METHOD PRIVATE DigitalMissingImageRejected
TEST('DigitalMissingImageRejected');
trustDigitalMissingImageRejected.cfg.restoreCommandOnRestart := TRUE;
trustDigitalMissingImageRejected.cfg.invert := TRUE;
trustDigitalMissingImageRejected.SeedSavedCommand(value := FALSE);
trustDigitalMissingImageRejected.simulatedBootDataLoaded := FALSE;
trustDigitalMissingImageRejected.simulatedOldBootData := FALSE;
trustDigitalMissingImageRejected();
AssertTrue(trustDigitalMissingImageRejected.sts.outputInhibited, 'Untrusted persistent image cannot restore output');
AssertFalse(trustDigitalMissingImageRejected.outSignal, 'Electrical output honors startup trust');
trustDigitalMissingImageRejected.simulatedBootDataLoaded := TRUE; trustDigitalMissingImageRejected.simulatedOldBootData := FALSE;
trustDigitalMissingImageRejected.SimulateStartup(); trustDigitalMissingImageRejected();
AssertTrue(trustDigitalMissingImageRejected.sts.outputInhibited, 'Later trust cannot revive previously rejected saved intent');
TEST_FINISHED();
END_METHOD

METHOD PRIVATE DigitalFreshCommandWithUntrustedImage
TEST('DigitalFreshCommandWithUntrustedImage');
trustDigitalFreshCommandWithUntrustedImage.cfg.restoreCommandOnRestart := TRUE;
trustDigitalFreshCommandWithUntrustedImage.cfg.invert := TRUE;
trustDigitalFreshCommandWithUntrustedImage.SeedSavedCommand(value := FALSE);
trustDigitalFreshCommandWithUntrustedImage.simulatedBootDataLoaded := TRUE;
trustDigitalFreshCommandWithUntrustedImage.simulatedOldBootData := TRUE;
trustDigitalFreshCommandWithUntrustedImage.SetOff();
trustDigitalFreshCommandWithUntrustedImage();
AssertFalse(trustDigitalFreshCommandWithUntrustedImage.sts.outputInhibited, 'Fresh command is independent of image trust');
AssertTrue(trustDigitalFreshCommandWithUntrustedImage.outSignal, 'Electrical output honors startup trust');
trustDigitalFreshCommandWithUntrustedImage.simulatedBootDataLoaded := TRUE; trustDigitalFreshCommandWithUntrustedImage.simulatedOldBootData := FALSE;
trustDigitalFreshCommandWithUntrustedImage.SimulateStartup(); trustDigitalFreshCommandWithUntrustedImage();
AssertFalse(trustDigitalFreshCommandWithUntrustedImage.sts.outputInhibited, 'Fresh command remains valid for later trusted restoration');
TEST_FINISHED();
END_METHOD

METHOD PRIVATE AnalogBackupImageRejected
TEST('AnalogBackupImageRejected');
trustAnalogBackupImageRejected.cfg.restoreCommandOnRestart := TRUE;
trustAnalogBackupImageRejected.cfg.useRawValue := TRUE; trustAnalogBackupImageRejected.cfg.safeRaw := 17.0;
trustAnalogBackupImageRejected.SeedSavedCommand(value := 42.0);
trustAnalogBackupImageRejected.simulatedBootDataLoaded := TRUE;
trustAnalogBackupImageRejected.simulatedOldBootData := TRUE;
trustAnalogBackupImageRejected();
AssertTrue(trustAnalogBackupImageRejected.sts.outputInhibited, 'Untrusted persistent image cannot restore output');
AssertEquals_REAL(17.0, trustAnalogBackupImageRejected.sts.rawReal, 0.001, 'Analog output honors startup trust');
trustAnalogBackupImageRejected.simulatedBootDataLoaded := TRUE; trustAnalogBackupImageRejected.simulatedOldBootData := FALSE;
trustAnalogBackupImageRejected.SimulateStartup(); trustAnalogBackupImageRejected();
AssertTrue(trustAnalogBackupImageRejected.sts.outputInhibited, 'Later trust cannot revive previously rejected saved intent');
TEST_FINISHED();
END_METHOD

METHOD PRIVATE AnalogMissingImageRejected
TEST('AnalogMissingImageRejected');
trustAnalogMissingImageRejected.cfg.restoreCommandOnRestart := TRUE;
trustAnalogMissingImageRejected.cfg.useRawValue := TRUE; trustAnalogMissingImageRejected.cfg.safeRaw := 17.0;
trustAnalogMissingImageRejected.SeedSavedCommand(value := 42.0);
trustAnalogMissingImageRejected.simulatedBootDataLoaded := FALSE;
trustAnalogMissingImageRejected.simulatedOldBootData := FALSE;
trustAnalogMissingImageRejected();
AssertTrue(trustAnalogMissingImageRejected.sts.outputInhibited, 'Untrusted persistent image cannot restore output');
AssertEquals_REAL(17.0, trustAnalogMissingImageRejected.sts.rawReal, 0.001, 'Analog output honors startup trust');
trustAnalogMissingImageRejected.simulatedBootDataLoaded := TRUE; trustAnalogMissingImageRejected.simulatedOldBootData := FALSE;
trustAnalogMissingImageRejected.SimulateStartup(); trustAnalogMissingImageRejected();
AssertTrue(trustAnalogMissingImageRejected.sts.outputInhibited, 'Later trust cannot revive previously rejected saved intent');
TEST_FINISHED();
END_METHOD

METHOD PRIVATE AnalogFreshCommandWithUntrustedImage
TEST('AnalogFreshCommandWithUntrustedImage');
trustAnalogFreshCommandWithUntrustedImage.cfg.restoreCommandOnRestart := TRUE;
trustAnalogFreshCommandWithUntrustedImage.cfg.useRawValue := TRUE; trustAnalogFreshCommandWithUntrustedImage.cfg.safeRaw := 17.0;
trustAnalogFreshCommandWithUntrustedImage.SeedSavedCommand(value := 42.0);
trustAnalogFreshCommandWithUntrustedImage.simulatedBootDataLoaded := TRUE;
trustAnalogFreshCommandWithUntrustedImage.simulatedOldBootData := TRUE;
trustAnalogFreshCommandWithUntrustedImage.SetValue(rValue := 42.0);
trustAnalogFreshCommandWithUntrustedImage();
AssertFalse(trustAnalogFreshCommandWithUntrustedImage.sts.outputInhibited, 'Fresh command is independent of image trust');
AssertEquals_REAL(42.0, trustAnalogFreshCommandWithUntrustedImage.sts.rawReal, 0.001, 'Analog output honors startup trust');
trustAnalogFreshCommandWithUntrustedImage.simulatedBootDataLoaded := TRUE; trustAnalogFreshCommandWithUntrustedImage.simulatedOldBootData := FALSE;
trustAnalogFreshCommandWithUntrustedImage.SimulateStartup(); trustAnalogFreshCommandWithUntrustedImage();
AssertFalse(trustAnalogFreshCommandWithUntrustedImage.sts.outputInhibited, 'Fresh command remains valid for later trusted restoration');
TEST_FINISHED();
END_METHOD

END_FUNCTION_BLOCK

// ---- Testing/POUs/FB_OutputRestart_Probe.TcPOU
// Injects a previously persisted value into an otherwise fresh instance.
// This tests startup policy, NOT actual TwinCAT persistent-image durability.
FUNCTION_BLOCK FB_OutputRestart_Probe EXTENDS TcForge.FB_DigitalOutput
VAR_INPUT
    simulatedBootDataLoaded : BOOL := TRUE;
    simulatedOldBootData : BOOL;
END_VAR

SUPER^();

METHOD PUBLIC SeedSavedCommand
VAR_INPUT
    value : BOOL;
END_VAR
_savedCommand := value;
_savedCommandValid := TRUE;
END_METHOD

// Policy probe: reset volatile arming only; not a runtime/persistent-image test.
METHOD PUBLIC SimulateStartup
_startup := TRUE;
_commandReceived := FALSE;
_armed := FALSE;
_forceSafe := FALSE;
_safeRequested := FALSE;
_requestSync := FALSE;
END_METHOD

METHOD PROTECTED _HasTrustedPersistentImage : BOOL
// Local probe inputs only: never mutate TwinCAT system information.
_HasTrustedPersistentImage := simulatedBootDataLoaded AND NOT simulatedOldBootData;
END_METHOD

END_FUNCTION_BLOCK

// ---- Testing/POUs/FB_AnalogOutputRestart_Probe.TcPOU
// Injects a previously persisted value into an otherwise fresh instance.
// This tests startup policy, NOT actual TwinCAT persistent-image durability.
FUNCTION_BLOCK FB_AnalogOutputRestart_Probe EXTENDS TcForge.FB_AnalogOutput
VAR_INPUT
    simulatedBootDataLoaded : BOOL := TRUE;
    simulatedOldBootData : BOOL;
END_VAR

SUPER^();

METHOD PUBLIC SeedSavedCommand
VAR_INPUT
    value : REAL;
END_VAR
_savedCommand := value;
_savedCommandValid := TRUE;
END_METHOD

// Policy probe: reset volatile arming only; not a runtime/persistent-image test.
METHOD PUBLIC SimulateStartup
_startup := TRUE;
_commandReceived := FALSE;
_armed := FALSE;
_forceSafe := FALSE;
_safeRequested := FALSE;
_requestSync := 0.0;
END_METHOD

METHOD PROTECTED _HasTrustedPersistentImage : BOOL
// Local probe inputs only: never mutate TwinCAT system information.
_HasTrustedPersistentImage := simulatedBootDataLoaded AND NOT simulatedOldBootData;
END_METHOD

END_FUNCTION_BLOCK

// ---- Testing/Tests/FB_IOQualityMonitor_Test.TcPOU
FUNCTION_BLOCK FB_IOQualityMonitor_Test EXTENDS TcUnit.FB_TestSuite
VAR
_done, _cyclicDone : BOOL;
_phase : UINT;
_stale : TcForge.FB_IOQualityMonitor;
_clock : TON;
_boundaryClock : TON;
_boundary : TcForge.FB_IOQualityMonitor;
_boundaryStarted, _boundaryDone : BOOL;
END_VAR

IF NOT _done THEN
StartupNeedsNewProducerSample();
CommunicationRecoveryNeedsNewSample();
DeviceAndInvalidSampleReject();
SequenceResetNeedsNewBaseline();
DisableRequiresReacquisition();
TimeoutConfigurationReacquires();
QualityRecoveryDoesNotRearmOutput();
EtherCATStateAndWorkingCounter();
_done := TRUE; END_IF;
CyclicFreshness();
FreshnessBoundary();

METHOD StartupNeedsNewProducerSample
VAR
fb : TcForge.FB_IOQualityMonitor;
outp : TcForge.FB_DigitalOutput;
bitIndex : INT;
mask : WORD;
END_VAR
TEST('StartupNeedsNewProducerSample');
fb(enabled := TRUE, communicationGood := TRUE, deviceGood := TRUE, sampleValid := TRUE, sampleSequence := 10);
AssertEquals_INT(Expected := 0, Actual := fb.quality, Message := 'First observed frame is only a baseline');
fb(sampleSequence := 11);
AssertEquals_INT(Expected := 2, Actual := fb.quality, Message := 'New coherent producer sample enables quality');
TEST_FINISHED();
END_METHOD

METHOD CommunicationRecoveryNeedsNewSample
VAR
fb : TcForge.FB_IOQualityMonitor;
outp : TcForge.FB_DigitalOutput;
bitIndex : INT;
mask : WORD;
END_VAR
TEST('CommunicationRecoveryNeedsNewSample');
fb(enabled := TRUE, communicationGood := TRUE, deviceGood := TRUE, sampleValid := TRUE, sampleSequence := 10); fb(sampleSequence := 11);
fb(communicationGood := FALSE);
AssertEquals_INT(Expected := 1, Actual := fb.quality, Message := 'Communication loss is immediate');
fb(communicationGood := TRUE);
AssertEquals_INT(Expected := 1, Actual := fb.quality, Message := 'Frozen sample cannot restore quality');
fb(sampleSequence := 12);
AssertEquals_INT(Expected := 2, Actual := fb.quality, Message := 'Fresh sample restores quality');
TEST_FINISHED();
END_METHOD

METHOD DeviceAndInvalidSampleReject
VAR
fb : TcForge.FB_IOQualityMonitor;
outp : TcForge.FB_DigitalOutput;
bitIndex : INT;
mask : WORD;
END_VAR
TEST('DeviceAndInvalidSampleReject');
fb(enabled := TRUE, communicationGood := TRUE, deviceGood := TRUE, sampleValid := TRUE, sampleSequence := 1); fb(sampleSequence := 2);
fb(deviceGood := FALSE);
AssertEquals_INT(Expected := 3, Actual := fb.reason, Message := 'Device fault is distinct');
fb(deviceGood := TRUE, sampleValid := FALSE, sampleSequence := 3);
AssertEquals_INT(Expected := 4, Actual := fb.reason, Message := 'Invalid frame is distinct');
fb(sampleValid := TRUE);
AssertEquals_INT(Expected := 1, Actual := fb.quality, Message := 'Previously invalid sample cannot become fresh');
fb(sampleSequence := 4);
AssertEquals_INT(Expected := 2, Actual := fb.quality, Message := 'Fresh valid update recovers');
TEST_FINISHED();
END_METHOD

METHOD SequenceResetNeedsNewBaseline
VAR
fb : TcForge.FB_IOQualityMonitor;
outp : TcForge.FB_DigitalOutput;
bitIndex : INT;
mask : WORD;
END_VAR
TEST('SequenceResetNeedsNewBaseline');
fb(enabled := TRUE, communicationGood := TRUE, deviceGood := TRUE, sampleValid := TRUE, sampleSequence := 10); fb(sampleSequence := 11);
fb(sampleSequence := 0);
AssertEquals_INT(Expected := 7, Actual := fb.reason, Message := 'Producer restart invalidates old session');
fb(); AssertEquals_INT(Expected := 1, Actual := fb.quality, Message := 'Repeated reset sequence stays bad');
fb(sampleSequence := 1); AssertEquals_INT(Expected := 2, Actual := fb.quality, Message := 'New producer update recovers');
TEST_FINISHED();
END_METHOD

METHOD DisableRequiresReacquisition
VAR
fb : TcForge.FB_IOQualityMonitor;
outp : TcForge.FB_DigitalOutput;
bitIndex : INT;
mask : WORD;
END_VAR
TEST('DisableRequiresReacquisition');
fb(enabled := TRUE, communicationGood := TRUE, deviceGood := TRUE, sampleValid := TRUE, sampleSequence := 1); fb(sampleSequence := 2);
fb(enabled := FALSE); fb(enabled := TRUE);
AssertEquals_INT(Expected := 0, Actual := fb.quality, Message := 'Reenable starts unqualified');
fb(sampleSequence := 3); AssertEquals_INT(Expected := 2, Actual := fb.quality, Message := 'New sample reacquires');
TEST_FINISHED();
END_METHOD

METHOD TimeoutConfigurationReacquires
VAR
fb : TcForge.FB_IOQualityMonitor;
outp : TcForge.FB_DigitalOutput;
bitIndex : INT;
mask : WORD;
END_VAR
TEST('TimeoutConfigurationReacquires');
fb(enabled := TRUE, communicationGood := TRUE, deviceGood := TRUE, sampleValid := TRUE, sampleSequence := 1); fb(sampleSequence := 2);
fb(timeout := T#0MS); AssertEquals_INT(Expected := 6, Actual := fb.reason, Message := 'Zero freshness deadline rejected');
fb(timeout := T#500MS); AssertFalse(Condition := fb.quality = TcForge.E_IO_Quality.GOOD, Message := 'Timeout edit cannot revive cached sample');
fb(sampleSequence := 3); AssertEquals_INT(Expected := 2, Actual := fb.quality, Message := 'Valid config and fresh sample recover');
TEST_FINISHED();
END_METHOD

METHOD QualityRecoveryDoesNotRearmOutput
VAR
fb : TcForge.FB_IOQualityMonitor;
outp : TcForge.FB_DigitalOutput;
bitIndex : INT;
mask : WORD;
END_VAR
TEST('QualityRecoveryDoesNotRearmOutput');
fb(enabled := TRUE, communicationGood := TRUE, deviceGood := TRUE, sampleValid := TRUE, sampleSequence := 1); fb(sampleSequence := 2);
outp(inpQuality := fb.quality); outp.SetOn(); outp(); AssertTrue(Condition := outp.outSignal, Message := 'Fixture energized');
fb(communicationGood := FALSE); outp(inpQuality := fb.quality);
fb(communicationGood := TRUE, sampleSequence := 3); outp(inpQuality := fb.quality);
AssertFalse(Condition := outp.outSignal, Message := 'Adapter cannot rearm retained output intent');
outp.SetOn(); outp(); AssertTrue(Condition := outp.outSignal, Message := 'Explicit command restores output');
TEST_FINISHED();
END_METHOD

METHOD EtherCATStateAndWorkingCounter
VAR
fb : TcForge.FB_IOQualityMonitor;
outp : TcForge.FB_DigitalOutput;
bitIndex : INT;
mask : WORD;
END_VAR
TEST('EtherCATStateAndWorkingCounter');
AssertTrue(Condition := TcForge.F_EtherCATSlaveDataValid(TRUE, FALSE, WORD#16#F008), Message := 'OP and port flags are healthy');
AssertFalse(Condition := TcForge.F_EtherCATSlaveDataValid(FALSE, FALSE, WORD#16#0008), Message := 'Unmapped diagnostics never qualify');
AssertFalse(Condition := TcForge.F_EtherCATSlaveDataValid(TRUE, TRUE, WORD#16#0008), Message := 'Working counter failure invalidates');
AssertFalse(Condition := TcForge.F_EtherCATSlaveDataValid(TRUE, FALSE, WORD#16#0004), Message := 'SAFEOP is not operational');
FOR bitIndex := 0 TO 15 DO
    mask := SHL(WORD#1, bitIndex);
    IF (mask AND WORD#16#0F30) <> WORD#0 THEN
        AssertFalse(Condition := TcForge.F_EtherCATSlaveDataValid(TRUE, FALSE, WORD#16#0008 OR mask), Message := 'Every documented error flag invalidates');
    END_IF;
END_FOR;
TEST_FINISHED();
END_METHOD

METHOD CyclicFreshness
IF _cyclicDone THEN RETURN; END_IF;
TEST('DuplicateProducerSamplesExpire');
CASE _phase OF
0:
    _stale(enabled := TRUE, communicationGood := TRUE, deviceGood := TRUE, sampleValid := TRUE, sampleSequence := 1, timeout := T#50MS);
    _stale(sampleSequence := 2);
    _phase := 1;
1:
    _clock(IN := TRUE, PT := T#150MS); _stale();
    IF _clock.Q THEN
        AssertEquals_INT(Expected := 1, Actual := _stale.quality, Message := 'Repeated valid value/frame does not refresh deadline');
        AssertEquals_INT(Expected := 5, Actual := _stale.reason, Message := 'Stale reason persists until fresh data');
        _clock(IN := FALSE); _phase := 2;
    END_IF;
2:
    _clock(IN := TRUE, PT := T#1S);
    _stale(sampleSequence := _stale.sampleSequence + 1);
    IF _stale.quality = TcForge.E_IO_Quality.GOOD OR _clock.Q THEN
        AssertEquals_INT(Expected := 2, Actual := _stale.quality, Message := 'New producer data recovers without signal-value change');
        _cyclicDone := TRUE; TEST_FINISHED();
    END_IF;
END_CASE;
END_METHOD

METHOD FreshnessBoundary
IF _boundaryDone THEN RETURN; END_IF;
TEST('FreshFrameAtDeadlineCannotHideExpiry');
IF NOT _boundaryStarted THEN
    _boundary(enabled := TRUE, communicationGood := TRUE, deviceGood := TRUE, sampleValid := TRUE, sampleSequence := 1, timeout := T#50MS);
    _boundary(sampleSequence := 2);
    _boundaryClock(IN := TRUE, PT := T#50MS);
    _boundaryStarted := TRUE;
ELSE
    _boundaryClock(IN := TRUE, PT := T#50MS);
    IF _boundaryClock.Q THEN
        _boundary(sampleSequence := 3);
        AssertEquals_INT(Expected := 5, Actual := _boundary.reason, Message := 'Late new frame cannot hide expired producer deadline');
        AssertEquals_INT(Expected := 1, Actual := _boundary.quality, Message := 'Deadline is measured from prior sample, not following scan');
        _boundaryDone := TRUE; TEST_FINISHED();
    ELSE
        _boundary();
    END_IF;
END_IF;
END_METHOD

END_FUNCTION_BLOCK

// ---- Testing/Tests/FB_InputLifecycle_Test.TcPOU
FUNCTION_BLOCK FB_InputLifecycle_Test EXTENDS TcUnit.FB_TestSuite
VAR
_done : BOOL;
_watchDone : BOOL;
_watch : TcForge.FB_DigitalInput;
_clock : TON;
END_VAR

IF NOT _done THEN
    InvalidInputTypeCannotPublishGood();
    RawBypassStillValidatesInputType();
    InvalidScalingFreezesFilterAndRecovers();
    UnknownQualityFreezesConditionedValue();
    InvalidConfigCannotReinterpretHeldRaw();
    RawBypassInvalidNumericConfigIsBad();
    _done := TRUE;
END_IF;
UnknownDigitalQualityExpiresWatchdog();

METHOD InvalidInputTypeCannotPublishGood
VAR
    fb : TcForge.FB_AnalogInput;
    held : REAL;
END_VAR
TEST('InvalidInputTypeCannotPublishGood');
fb.cfg.inputType := __SYSTEM.TYPE_CLASS.TYPE_REAL;
fb.cfg.rawMax := 100.0;
fb.inRaw.fReal := 80.0;
fb();
held := fb.sts.value;
fb.cfg.inputType := __SYSTEM.TYPE_CLASS.TYPE_BOOL;
fb.inRaw.fReal := 20.0;
fb();
AssertEquals_DINT(Expected := TcForge.E_AnalogInput_Fault.BadConfig, Actual := fb.GetFaultCode(), Message := 'Unsupported input interpretation faults immediately');
AssertEquals_DINT(Expected := TcForge.E_IO_Quality.BAD, Actual := fb.sts.quality, Message := 'Unsupported interpretation cannot advertise usable quality');
AssertTrue(Condition := fb.sts.value = held AND fb.sts.rawReal = 80.0, Message := 'Invalid interpretation preserves last usable values');
fb.cfg.inputType := __SYSTEM.TYPE_CLASS.TYPE_REAL;
fb();
AssertFalse(Condition := fb.IsFaulted(), Message := 'Input configuration recovery is automatic');
AssertTrue(Condition := ABS(fb.sts.value - 20.0) < 0.001, Message := 'Recovered interpretation consumes fresh sample');
TEST_FINISHED();
END_METHOD

METHOD RawBypassStillValidatesInputType
VAR
    fb : TcForge.FB_AnalogInput;
    held : REAL;
END_VAR
TEST('RawBypassStillValidatesInputType');
fb.cfg.useRawValue := TRUE;
fb.cfg.inputType := __SYSTEM.TYPE_CLASS.TYPE_BOOL;
fb.inRaw.fReal := 90.0;
fb();
AssertTrue(Condition := fb.IsFaulted(), Message := 'Raw bypass cannot bypass type validation');
AssertEquals_DINT(Expected := TcForge.E_IO_Quality.BAD, Actual := fb.sts.quality, Message := 'Invalid startup is BAD');
AssertTrue(Condition := fb.sts.value = 0.0, Message := 'Invalid first scan publishes no fabricated value');
TEST_FINISHED();
END_METHOD

METHOD InvalidScalingFreezesFilterAndRecovers
VAR
    fb : TcForge.FB_AnalogInput;
    held : REAL;
END_VAR
TEST('InvalidScalingFreezesFilterAndRecovers');
fb.cfg.inputType := __SYSTEM.TYPE_CLASS.TYPE_REAL;
fb.cfg.rawMax := 100.0;
fb.inRaw.fReal := 80.0;
fb();
held := fb.sts.value;
fb.cfg.filterTau := T#1S;
fb.cfg.rawMax := fb.cfg.rawMin;
fb.inRaw.fReal := 0.0;
fb(); fb(); fb();
AssertTrue(Condition := fb.sts.value = held, Message := 'Invalid scaling cannot move the conditioned output');
AssertEquals_DINT(Expected := TcForge.E_IO_Quality.BAD, Actual := fb.sts.quality, Message := 'Invalid scaling is BAD');
fb.cfg.rawMax := 100.0;
fb.inRaw.fReal := 80.0;
fb();
AssertFalse(Condition := fb.IsFaulted(), Message := 'Valid scaling clears configuration fault');
AssertTrue(Condition := fb.sts.value = held, Message := 'Enabling filtering after prior data reseeds from first valid sample');
TEST_FINISHED();
END_METHOD

METHOD UnknownQualityFreezesConditionedValue
VAR
    fb : TcForge.FB_AnalogInput;
    held : REAL;
END_VAR
TEST('UnknownQualityFreezesConditionedValue');
fb.cfg.inputType := __SYSTEM.TYPE_CLASS.TYPE_REAL;
fb.cfg.rawMax := 100.0;
fb.inRaw.fReal := 80.0;
fb.cfg.filterTau := T#1S;
fb();
held := fb.sts.value;
fb.inRaw.fReal := 100.0;
fb(inpQuality := TcForge.E_IO_Quality.UNKNOWN);
fb(); fb();
AssertTrue(Condition := fb.sts.value = held AND fb.sts.rawReal = 80.0, Message := 'Unavailable sample cannot advance the filter');
fb(inpQuality := TcForge.E_IO_Quality.GOOD);
AssertTrue(Condition := fb.sts.value > held, Message := 'A fresh valid sample resumes conditioning');
TEST_FINISHED();
END_METHOD

METHOD InvalidConfigCannotReinterpretHeldRaw
VAR
    fb : TcForge.FB_AnalogInput;
    held : REAL;
END_VAR
TEST('InvalidConfigCannotReinterpretHeldRaw');
fb.cfg.inputType := __SYSTEM.TYPE_CLASS.TYPE_REAL;
fb.cfg.rawMax := 100.0;
fb.inRaw.fReal := 80.0;
fb();
held := fb.sts.value;
fb.cfg.euMax := 200.0;
fb.inRaw.fReal := 20.0;
fb(inpQuality := TcForge.E_IO_Quality.BAD);
AssertTrue(Condition := fb.sts.value = held AND fb.sts.scaled = held, Message := 'No fresh sample means no reinterpretation under new scaling');
fb(inpQuality := TcForge.E_IO_Quality.GOOD);
AssertTrue(Condition := ABS(fb.sts.value - 40.0) < 0.001, Message := 'Valid fresh sample uses current scaling');
TEST_FINISHED();
END_METHOD

METHOD RawBypassInvalidNumericConfigIsBad
VAR
    fb : TcForge.FB_AnalogInput;
    held : REAL;
    invalid : TcForge.U_IoRaw_In;
END_VAR
TEST('RawBypassInvalidNumericConfigIsBad');
fb.cfg.useRawValue := TRUE;
fb.cfg.inputType := __SYSTEM.TYPE_CLASS.TYPE_REAL;
fb.inRaw.fReal := 7.0;
fb();
held := fb.sts.value;
// Infinity via raw IEEE-754 bits, avoiding invalid arithmetic in the test.
invalid.dw := DWORD#16#7F800000;
fb.cfg.euMax := invalid.fReal;
fb.inRaw.fReal := 9.0;
fb();
AssertTrue(Condition := fb.IsFaulted(), Message := 'Nonfinite config rejected in bypass too');
AssertEquals_DINT(Expected := TcForge.E_IO_Quality.BAD, Actual := fb.sts.quality, Message := 'Config fault cannot retain GOOD in bypass');
AssertTrue(Condition := fb.sts.value = held, Message := 'Invalid numeric config holds last value');
TEST_FINISHED();
END_METHOD

METHOD UnknownDigitalQualityExpiresWatchdog
IF _watchDone THEN RETURN; END_IF;
TEST('UnknownDigitalQualityExpiresWatchdog');
_watch.cfg.qualityFaultAfter := T#30MS;
_watch(inpQuality := TcForge.E_IO_Quality.UNKNOWN);
_clock(IN := TRUE, PT := T#100MS);
IF _clock.Q THEN
    AssertEquals_DINT(Expected := TcForge.E_DigitalInput_Fault.BadQuality, Actual := _watch.GetFaultCode(), Message := 'Missing input source expires the configured watchdog');
    _watch.Reset();
    _watch(inpQuality := TcForge.E_IO_Quality.GOOD, inSignal := TRUE);
    AssertFalse(Condition := _watch.IsFaulted(), Message := 'Healthy source with explicit reset recovers');
    AssertTrue(Condition := _watch.sts.value, Message := 'Recovered source consumes fresh digital input');
    _watchDone := TRUE;
    TEST_FINISHED();
END_IF;
END_METHOD

END_FUNCTION_BLOCK

// ---- Testing/Tests/FB_OperatorMailbox_Test.TcPOU
FUNCTION_BLOCK FB_OperatorMailbox_Test EXTENDS TcUnit.FB_TestSuite
VAR
 extra0 : TcForge.FB_AnalogOutput;
 extra1 : TcForge.FB_TwoPosActuator;
 extra2 : TcForge.FB_StateMachine;
 extra3 : TcForge.FB_StateMachine;
 extra4 : TcForge.FB_AlarmSimple;
 extra5 : TcForge.FB_AlarmLimit;
 done : BOOL;
 rsp : TcForge.E_RpcMethodResponse;
 ready : BOOL;
 cmd : TcForge.E_OperatorCommand;
 i : INT;
 box0 : TcForge.FB_OperatorMailbox;
 device0 : TcForge.FB_DigitalOutput;
 box1 : TcForge.FB_OperatorMailbox;
 device1 : TcForge.FB_DigitalOutput;
 box2 : TcForge.FB_OperatorMailbox;
 device2 : TcForge.FB_DigitalOutput;
 box3 : TcForge.FB_OperatorMailbox;
 device3 : TcForge.FB_DigitalOutput;
 box4 : TcForge.FB_OperatorMailbox;
 device4 : TcForge.FB_DigitalOutput;
 box5 : TcForge.FB_OperatorMailbox;
 device5 : TcForge.FB_DigitalOutput;
 box6 : TcForge.FB_OperatorMailbox;
 device6 : TcForge.FB_DigitalOutput;
 box7 : TcForge.FB_OperatorMailbox;
 device7 : TcForge.FB_DigitalOutput;
 box8 : TcForge.FB_OperatorMailbox;
 device8 : TcForge.FB_DigitalOutput;
 box9 : TcForge.FB_OperatorMailbox;
 device9 : TcForge.FB_DigitalOutput;
 box10 : TcForge.FB_OperatorMailbox;
 device10 : TcForge.FB_DigitalOutput;
 box11 : TcForge.FB_OperatorMailbox;
 device11 : TcForge.FB_DigitalOutput;
 box12 : TcForge.FB_OperatorMailbox;
 device12 : TcForge.FB_DigitalOutput;
END_VAR

IF done THEN RETURN; END_IF;
RejectBeforeOwner();
RejectZeroId();
RejectDuplicate();
BoundedAdmission();
AbortCancelsStart();
StopCannotReplaceAbort();
DispatchExcludesRpc();
ProgramBarrierCancelsNormal();
ProgramBarrierPreservesUrgent();
BoundedResultRetention();
OwnerDispatchChangesOutput();
OwnerRechecksSourceLock();
ProgramSafeCancelsQueuedOn();
AnalogOwnerDispatch();
ActuatorOwnerDispatch();
SequenceOwnerDispatch();
InheritedResetUsesConcreteOverride();
AlarmOwnerDispatch();
CompositeAlarmOwnerDispatch();
done := TRUE;

METHOD RejectBeforeOwner
TEST('RejectBeforeOwner');
rsp := box0.Submit(1, TcForge.E_OperatorCommand.SetOn, 0);
Check(TcForge.E_RpcMethodResponse.REJECTED_NOT_READY);
TEST_FINISHED();
END_METHOD

METHOD RejectZeroId
TEST('RejectZeroId');
ready := box1.BeginConsume(); rsp := box1.Submit(0, TcForge.E_OperatorCommand.SetOn, 0);
Check(TcForge.E_RpcMethodResponse.REJECTED_INVALID_PARAMETER);
TEST_FINISHED();
END_METHOD

METHOD RejectDuplicate
TEST('RejectDuplicate');
ready := box2.BeginConsume(); rsp := box2.Submit(1, TcForge.E_OperatorCommand.SetOn, 0); rsp := box2.Submit(1, TcForge.E_OperatorCommand.Abort, 0);
Check(TcForge.E_RpcMethodResponse.REJECTED_DUPLICATE_REQUEST);
TEST_FINISHED();
END_METHOD

METHOD BoundedAdmission
TEST('BoundedAdmission');
ready := box3.BeginConsume(); rsp := box3.Submit(1, TcForge.E_OperatorCommand.SetOn, 0); Check(TcForge.E_RpcMethodResponse.QUEUED); rsp := box3.Submit(2, TcForge.E_OperatorCommand.SetOn, 0); Check(TcForge.E_RpcMethodResponse.REJECTED_BUSY);
TEST_FINISHED();
END_METHOD

METHOD AbortCancelsStart
TEST('AbortCancelsStart');
ready := box4.BeginConsume(); rsp := box4.Submit(1, TcForge.E_OperatorCommand.Start, 0); rsp := box4.Submit(2, TcForge.E_OperatorCommand.Abort, 0); Check(TcForge.E_RpcMethodResponse.QUEUED); rsp := box4.GetResult(1); Check(TcForge.E_RpcMethodResponse.CANCELLED); ready := box4.BeginConsume(command => cmd); AssertTrue(ready, 'Abort available'); AssertEquals_DINT(TcForge.E_OperatorCommand.Abort, cmd, 'Urgent command selected'); box4.EndConsume(TcForge.E_RpcMethodResponse.ACCEPTED);
TEST_FINISHED();
END_METHOD

METHOD StopCannotReplaceAbort
TEST('StopCannotReplaceAbort');
ready := box5.BeginConsume(); rsp := box5.Submit(1, TcForge.E_OperatorCommand.Abort, 0); rsp := box5.Submit(2, TcForge.E_OperatorCommand.Stop, 0); Check(TcForge.E_RpcMethodResponse.REJECTED_BUSY);
TEST_FINISHED();
END_METHOD

METHOD DispatchExcludesRpc
TEST('DispatchExcludesRpc');
ready := box6.BeginConsume(); rsp := box6.Submit(1, TcForge.E_OperatorCommand.SetOn, 0); ready := box6.BeginConsume(); rsp := box6.Submit(2, TcForge.E_OperatorCommand.Abort, 0); Check(TcForge.E_RpcMethodResponse.REJECTED_BUSY); rsp := box6.GetResult(1); Check(TcForge.E_RpcMethodResponse.REJECTED_BUSY); box6.EndConsume(TcForge.E_RpcMethodResponse.REJECTED_FAULTED); rsp := box6.GetResult(1); Check(TcForge.E_RpcMethodResponse.REJECTED_FAULTED); AssertEquals_DINT(box6.ownerTask, box6.lastExecutionTask, 'Only owning task executed');
TEST_FINISHED();
END_METHOD

METHOD ProgramBarrierCancelsNormal
TEST('ProgramBarrierCancelsNormal');
ready := box7.BeginConsume(); rsp := box7.Submit(1, TcForge.E_OperatorCommand.Start, 0); box7.CancelNormal(); ready := box7.BeginConsume(); AssertFalse(ready, 'Cancelled normal command cannot execute'); rsp := box7.GetResult(1); Check(TcForge.E_RpcMethodResponse.CANCELLED);
TEST_FINISHED();
END_METHOD

METHOD ProgramBarrierPreservesUrgent
TEST('ProgramBarrierPreservesUrgent');
ready := box8.BeginConsume(); box8.CancelNormal(); rsp := box8.Submit(1, TcForge.E_OperatorCommand.Start, 0); Check(TcForge.E_RpcMethodResponse.REJECTED_BUSY); rsp := box8.Submit(2, TcForge.E_OperatorCommand.Abort, 0); Check(TcForge.E_RpcMethodResponse.QUEUED); ready := box8.BeginConsume(); AssertTrue(ready, 'Abort survives barrier'); box8.EndConsume(TcForge.E_RpcMethodResponse.ACCEPTED);
TEST_FINISHED();
END_METHOD

METHOD BoundedResultRetention
TEST('BoundedResultRetention');
ready := box9.BeginConsume(); FOR i := 1 TO 9 DO rsp := box9.Submit(INT_TO_ULINT(i), TcForge.E_OperatorCommand.SetOn, 0); ready := box9.BeginConsume(); box9.EndConsume(TcForge.E_RpcMethodResponse.ACCEPTED); END_FOR; rsp := box9.GetResult(1); Check(TcForge.E_RpcMethodResponse.REJECTED_UNKNOWN_REQUEST); rsp := box9.GetResult(2); Check(TcForge.E_RpcMethodResponse.ACCEPTED); rsp := box9.GetResult(9); Check(TcForge.E_RpcMethodResponse.ACCEPTED);
TEST_FINISHED();
END_METHOD

METHOD OwnerDispatchChangesOutput
TEST('OwnerDispatchChangesOutput');
device10(); rsp := device10.OperatorSetOn(1); Check(TcForge.E_RpcMethodResponse.QUEUED); AssertFalse(device10.outSignal, 'RPC admission cannot energize'); device10(); AssertTrue(device10.outSignal, 'Owner executes accepted output'); rsp := device10.OperatorCommandResult(1); Check(TcForge.E_RpcMethodResponse.ACCEPTED);
TEST_FINISHED();
END_METHOD

METHOD OwnerRechecksSourceLock
TEST('OwnerRechecksSourceLock');
device11(); rsp := device11.OperatorSetOn(1); device11.LockSource(TRUE); device11(); rsp := device11.OperatorCommandResult(1); Check(TcForge.E_RpcMethodResponse.REJECTED_SOURCE_NOT_ALLOWED); AssertFalse(device11.outSignal, 'Lock applied after submission blocks execution');
TEST_FINISHED();
END_METHOD

METHOD ProgramSafeCancelsQueuedOn
TEST('ProgramSafeCancelsQueuedOn');
device12(); rsp := device12.OperatorSetOn(1); device12.ForceSafe(); device12(); rsp := device12.OperatorCommandResult(1); Check(TcForge.E_RpcMethodResponse.CANCELLED); AssertFalse(device12.outSignal, 'Queued command cannot undo program shutdown');
TEST_FINISHED();
END_METHOD

METHOD PRIVATE Check
VAR_INPUT expected : TcForge.E_RpcMethodResponse; END_VAR
AssertEquals_DINT(expected, rsp, 'Mailbox response');
END_METHOD

METHOD AnalogOwnerDispatch
TEST('AnalogOwnerDispatch');
extra0(); rsp := extra0.OperatorSetValue(rValue := 25.0, requestId := 1); Check(TcForge.E_RpcMethodResponse.QUEUED); extra0(); rsp := extra0.OperatorCommandResult(1); Check(TcForge.E_RpcMethodResponse.ACCEPTED); AssertEquals_REAL(25.0, extra0.sts.commanded, 0.001, 'Analog value crosses mailbox');
TEST_FINISHED();
END_METHOD

METHOD ActuatorOwnerDispatch
TEST('ActuatorOwnerDispatch');
extra1(inRetracted := TRUE); rsp := extra1.OperatorAdvance(1); extra1(); rsp := extra1.OperatorCommandResult(1); Check(TcForge.E_RpcMethodResponse.ACCEPTED); AssertTrue(extra1.outAdvance, 'Owner starts actuator'); rsp := extra1.OperatorAbort(2); extra1(); AssertFalse(extra1.outAdvance OR extra1.outRetract, 'Remote abort drops both coils');
TEST_FINISHED();
END_METHOD

METHOD SequenceOwnerDispatch
TEST('SequenceOwnerDispatch');
extra2(); rsp := extra2.OperatorHome(1); extra2(); rsp := extra2.OperatorCommandResult(1); Check(TcForge.E_RpcMethodResponse.ACCEPTED); AssertEquals_DINT(TcForge.E_SM_State.HOMING, extra2.Status.State, 'Owner starts homing');
TEST_FINISHED();
END_METHOD

METHOD InheritedResetUsesConcreteOverride
TEST('InheritedResetUsesConcreteOverride');
extra3(); extra3.Home(); extra3(); rsp := extra3.OperatorReset(1); extra3(); rsp := extra3.OperatorCommandResult(1); Check(TcForge.E_RpcMethodResponse.REJECTED_WRONG_STATE); AssertEquals_DINT(TcForge.E_SM_State.HOMING, extra3.Status.State, 'Base RPC does not bypass concrete Reset');
TEST_FINISHED();
END_METHOD

METHOD AlarmOwnerDispatch
TEST('AlarmOwnerDispatch');
extra4.cfg.common.bEnable := TRUE; extra4.cfg.common.bRequireAck := TRUE; extra4(inpActive := TRUE); extra4(inpActive := FALSE); AssertTrue(extra4.sts.latched, 'Alarm latched before RPC'); rsp := extra4.OperatorAck(1); extra4(); rsp := extra4.OperatorCommandResult(1); Check(TcForge.E_RpcMethodResponse.ACCEPTED); AssertFalse(extra4.sts.active, 'Owner acknowledges cleared alarm');
TEST_FINISHED();
END_METHOD

METHOD CompositeAlarmOwnerDispatch
TEST('CompositeAlarmOwnerDispatch');
extra5.cfg.Hi.common.bEnable := TRUE; extra5.cfg.Hi.common.bRequireAck := TRUE; extra5.cfg.Hi.bFailHigh := TRUE; extra5(inpPv := 10.0); extra5(inpPv := 0.0); AssertTrue(extra5.sts.Hi.latched, 'Composite alarm latched before RPC'); rsp := extra5.OperatorAck(1); extra5(); rsp := extra5.OperatorCommandResult(1); Check(TcForge.E_RpcMethodResponse.ACCEPTED); AssertFalse(extra5.sts.Hi.active, 'Owner acknowledges composite alarm');
TEST_FINISHED();
END_METHOD

END_FUNCTION_BLOCK

// ---- Testing/Tests/FB_CommandValidation_Test.TcPOU
FUNCTION_BLOCK FB_CommandValidation_Test EXTENDS TcUnit.FB_TestSuite
VAR
    done : BOOL;
    raw : DINT := 99;
    invalid : POINTER TO TcForge.E_Requester;
    rsp : TcForge.E_RpcMethodResponse;
    device0 : FB_StateMachine_Probe;
    device1 : FB_StateMachine_Probe;
    device2 : FB_StateMachine_Probe;
    device3 : FB_StateMachine_Probe;
    device4 : FB_StateMachine_Probe;
    device5 : FB_StateMachine_Probe;
    device6 : FB_StateMachine_Probe;
    device7 : FB_StateMachine_Probe;
    device8 : TcForge.FB_TwoPosActuator;
    device9 : TcForge.FB_TwoPosActuator;
    device10 : TcForge.FB_TwoPosActuator;
    device11 : TcForge.FB_TwoPosActuator;
    device12 : TcForge.FB_DigitalOutput;
    device13 : TcForge.FB_DigitalOutput;
    device14 : TcForge.FB_DigitalOutput;
    device15 : TcForge.FB_DigitalOutput;
    device16 : TcForge.FB_AnalogOutput;
    device17 : TcForge.FB_AnalogOutput;
    device18 : TcForge.FB_AnalogOutput;
    device19 : FB_DeviceBase_Probe;
    device20 : TcForge.FB_AlarmSimple;
    device21 : TcForge.FB_AlarmLimit;
END_VAR

IF done THEN RETURN; END_IF;
invalid := ADR(raw);
SequenceHomeRejectsInvalidIdentity();
SequenceStartRejectsInvalidIdentity();
SequencePauseRejectsInvalidIdentity();
SequenceProceedRejectsInvalidIdentity();
SequenceRetryRejectsInvalidIdentity();
SequenceStopRejectsInvalidIdentity();
SequenceAbortRejectsInvalidIdentity();
SequenceResetRejectsInvalidIdentity();
ActuatorAdvanceRejectsInvalidIdentity();
ActuatorRetractRejectsInvalidIdentity();
ActuatorAbortRejectsInvalidIdentity();
ActuatorResetRejectsInvalidIdentity();
DigitalSetOnRejectsInvalidIdentity();
DigitalSetOffRejectsInvalidIdentity();
DigitalForceSafeRejectsInvalidIdentity();
DigitalResetRejectsInvalidIdentity();
AnalogSetValueRejectsInvalidIdentity();
AnalogForceSafeRejectsInvalidIdentity();
AnalogResetRejectsInvalidIdentity();
BaseResetRejectsInvalidIdentity();
AlarmAckRejectsInvalidIdentity();
LimitAlarmAckRejectsInvalidIdentity();
done := TRUE;

METHOD SequenceHomeRejectsInvalidIdentity
TEST('SequenceHomeRejectsInvalidIdentity');
device0.ResetAll(); device0(); rsp := device0.Home();
AssertEquals_DINT(Expected := TcForge.E_RpcMethodResponse.ACCEPTED, Actual := rsp, Message := 'Valid Home queued before rejected request');
rsp := device0.Home(eRequester := invalid^);
AssertEquals_DINT(Expected := TcForge.E_RpcMethodResponse.REJECTED_INVALID_PARAMETER, Actual := rsp, Message := 'Invalid identity must reject before device-specific logic');
device0();
AssertEquals_DINT(Expected := TcForge.E_SM_State.HOMING, Actual := device0.Status.State, Message := 'Rejected request preserves queued Home');
TEST_FINISHED();
END_METHOD

METHOD SequenceStartRejectsInvalidIdentity
TEST('SequenceStartRejectsInvalidIdentity');
device1.ResetAll(); device1(); rsp := device1.Home();
AssertEquals_DINT(Expected := TcForge.E_RpcMethodResponse.ACCEPTED, Actual := rsp, Message := 'Valid Home queued before rejected request');
rsp := device1.Start(eRequester := invalid^);
AssertEquals_DINT(Expected := TcForge.E_RpcMethodResponse.REJECTED_INVALID_PARAMETER, Actual := rsp, Message := 'Invalid identity must reject before device-specific logic');
device1();
AssertEquals_DINT(Expected := TcForge.E_SM_State.HOMING, Actual := device1.Status.State, Message := 'Rejected request preserves queued Home');
TEST_FINISHED();
END_METHOD

METHOD SequencePauseRejectsInvalidIdentity
TEST('SequencePauseRejectsInvalidIdentity');
device2.ResetAll(); device2(); rsp := device2.Home();
AssertEquals_DINT(Expected := TcForge.E_RpcMethodResponse.ACCEPTED, Actual := rsp, Message := 'Valid Home queued before rejected request');
rsp := device2.Pause(eRequester := invalid^);
AssertEquals_DINT(Expected := TcForge.E_RpcMethodResponse.REJECTED_INVALID_PARAMETER, Actual := rsp, Message := 'Invalid identity must reject before device-specific logic');
device2();
AssertEquals_DINT(Expected := TcForge.E_SM_State.HOMING, Actual := device2.Status.State, Message := 'Rejected request preserves queued Home');
TEST_FINISHED();
END_METHOD

METHOD SequenceProceedRejectsInvalidIdentity
TEST('SequenceProceedRejectsInvalidIdentity');
device3.ResetAll(); device3(); rsp := device3.Home();
AssertEquals_DINT(Expected := TcForge.E_RpcMethodResponse.ACCEPTED, Actual := rsp, Message := 'Valid Home queued before rejected request');
rsp := device3.Proceed(eRequester := invalid^);
AssertEquals_DINT(Expected := TcForge.E_RpcMethodResponse.REJECTED_INVALID_PARAMETER, Actual := rsp, Message := 'Invalid identity must reject before device-specific logic');
device3();
AssertEquals_DINT(Expected := TcForge.E_SM_State.HOMING, Actual := device3.Status.State, Message := 'Rejected request preserves queued Home');
TEST_FINISHED();
END_METHOD

METHOD SequenceRetryRejectsInvalidIdentity
TEST('SequenceRetryRejectsInvalidIdentity');
device4.ResetAll(); device4(); rsp := device4.Home();
AssertEquals_DINT(Expected := TcForge.E_RpcMethodResponse.ACCEPTED, Actual := rsp, Message := 'Valid Home queued before rejected request');
rsp := device4.Retry(eRequester := invalid^);
AssertEquals_DINT(Expected := TcForge.E_RpcMethodResponse.REJECTED_INVALID_PARAMETER, Actual := rsp, Message := 'Invalid identity must reject before device-specific logic');
device4();
AssertEquals_DINT(Expected := TcForge.E_SM_State.HOMING, Actual := device4.Status.State, Message := 'Rejected request preserves queued Home');
TEST_FINISHED();
END_METHOD

METHOD SequenceStopRejectsInvalidIdentity
TEST('SequenceStopRejectsInvalidIdentity');
device5.ResetAll(); device5(); rsp := device5.Home();
AssertEquals_DINT(Expected := TcForge.E_RpcMethodResponse.ACCEPTED, Actual := rsp, Message := 'Valid Home queued before rejected request');
rsp := device5.Stop(eRequester := invalid^);
AssertEquals_DINT(Expected := TcForge.E_RpcMethodResponse.REJECTED_INVALID_PARAMETER, Actual := rsp, Message := 'Invalid identity must reject before device-specific logic');
device5();
AssertEquals_DINT(Expected := TcForge.E_SM_State.HOMING, Actual := device5.Status.State, Message := 'Rejected request preserves queued Home');
TEST_FINISHED();
END_METHOD

METHOD SequenceAbortRejectsInvalidIdentity
TEST('SequenceAbortRejectsInvalidIdentity');
device6.ResetAll(); device6(); rsp := device6.Home();
AssertEquals_DINT(Expected := TcForge.E_RpcMethodResponse.ACCEPTED, Actual := rsp, Message := 'Valid Home queued before rejected request');
rsp := device6.Abort(eRequester := invalid^);
AssertEquals_DINT(Expected := TcForge.E_RpcMethodResponse.REJECTED_INVALID_PARAMETER, Actual := rsp, Message := 'Invalid identity must reject before device-specific logic');
device6();
AssertEquals_DINT(Expected := TcForge.E_SM_State.HOMING, Actual := device6.Status.State, Message := 'Rejected request preserves queued Home');
TEST_FINISHED();
END_METHOD

METHOD SequenceResetRejectsInvalidIdentity
TEST('SequenceResetRejectsInvalidIdentity');
device7.ResetAll(); device7(); rsp := device7.Home();
AssertEquals_DINT(Expected := TcForge.E_RpcMethodResponse.ACCEPTED, Actual := rsp, Message := 'Valid Home queued before rejected request');
rsp := device7.Reset(eRequester := invalid^);
AssertEquals_DINT(Expected := TcForge.E_RpcMethodResponse.REJECTED_INVALID_PARAMETER, Actual := rsp, Message := 'Invalid identity must reject before device-specific logic');
device7();
AssertEquals_DINT(Expected := TcForge.E_SM_State.HOMING, Actual := device7.Status.State, Message := 'Rejected request preserves queued Home');
TEST_FINISHED();
END_METHOD

METHOD ActuatorAdvanceRejectsInvalidIdentity
TEST('ActuatorAdvanceRejectsInvalidIdentity');
device8(inRetracted := TRUE); device8.Advance(); device8();
rsp := device8.Advance(eRequester := invalid^);
AssertEquals_DINT(Expected := TcForge.E_RpcMethodResponse.REJECTED_INVALID_PARAMETER, Actual := rsp, Message := 'Invalid identity must reject before device-specific logic');
device8();
AssertTrue(Condition := device8.outAdvance AND NOT device8.outRetract, Message := 'Rejected command cannot change motion');
TEST_FINISHED();
END_METHOD

METHOD ActuatorRetractRejectsInvalidIdentity
TEST('ActuatorRetractRejectsInvalidIdentity');
device9(inRetracted := TRUE); device9.Advance(); device9();
rsp := device9.Retract(eRequester := invalid^);
AssertEquals_DINT(Expected := TcForge.E_RpcMethodResponse.REJECTED_INVALID_PARAMETER, Actual := rsp, Message := 'Invalid identity must reject before device-specific logic');
device9();
AssertTrue(Condition := device9.outAdvance AND NOT device9.outRetract, Message := 'Rejected command cannot change motion');
TEST_FINISHED();
END_METHOD

METHOD ActuatorAbortRejectsInvalidIdentity
TEST('ActuatorAbortRejectsInvalidIdentity');
device10(inRetracted := TRUE); device10.Advance(); device10();
rsp := device10.Abort(eRequester := invalid^);
AssertEquals_DINT(Expected := TcForge.E_RpcMethodResponse.REJECTED_INVALID_PARAMETER, Actual := rsp, Message := 'Invalid identity must reject before device-specific logic');
device10();
AssertTrue(Condition := device10.outAdvance AND NOT device10.outRetract, Message := 'Rejected command cannot change motion');
TEST_FINISHED();
END_METHOD

METHOD ActuatorResetRejectsInvalidIdentity
TEST('ActuatorResetRejectsInvalidIdentity');
device11(inRetracted := TRUE); device11.Advance(); device11();
rsp := device11.Reset(eRequester := invalid^);
AssertEquals_DINT(Expected := TcForge.E_RpcMethodResponse.REJECTED_INVALID_PARAMETER, Actual := rsp, Message := 'Invalid identity must reject before device-specific logic');
device11();
AssertTrue(Condition := device11.outAdvance AND NOT device11.outRetract, Message := 'Rejected command cannot change motion');
TEST_FINISHED();
END_METHOD

METHOD DigitalSetOnRejectsInvalidIdentity
TEST('DigitalSetOnRejectsInvalidIdentity');
device12();
rsp := device12.SetOn(eRequester := invalid^);
AssertEquals_DINT(Expected := TcForge.E_RpcMethodResponse.REJECTED_INVALID_PARAMETER, Actual := rsp, Message := 'Invalid identity must reject before device-specific logic');
device12();
AssertTrue(Condition := NOT device12.outSignal, Message := 'Rejected command cannot change output intent');
TEST_FINISHED();
END_METHOD

METHOD DigitalSetOffRejectsInvalidIdentity
TEST('DigitalSetOffRejectsInvalidIdentity');
device13.SetOn(); device13();
rsp := device13.SetOff(eRequester := invalid^);
AssertEquals_DINT(Expected := TcForge.E_RpcMethodResponse.REJECTED_INVALID_PARAMETER, Actual := rsp, Message := 'Invalid identity must reject before device-specific logic');
device13();
AssertTrue(Condition := device13.outSignal, Message := 'Rejected command cannot change output intent');
TEST_FINISHED();
END_METHOD

METHOD DigitalForceSafeRejectsInvalidIdentity
TEST('DigitalForceSafeRejectsInvalidIdentity');
device14.SetOn(); device14();
rsp := device14.ForceSafe(eRequester := invalid^);
AssertEquals_DINT(Expected := TcForge.E_RpcMethodResponse.REJECTED_INVALID_PARAMETER, Actual := rsp, Message := 'Invalid identity must reject before device-specific logic');
device14();
AssertTrue(Condition := device14.outSignal, Message := 'Rejected command cannot change output intent');
TEST_FINISHED();
END_METHOD

METHOD DigitalResetRejectsInvalidIdentity
TEST('DigitalResetRejectsInvalidIdentity');
device15.SetOn(); device15();
rsp := device15.Reset(eRequester := invalid^);
AssertEquals_DINT(Expected := TcForge.E_RpcMethodResponse.REJECTED_INVALID_PARAMETER, Actual := rsp, Message := 'Invalid identity must reject before device-specific logic');
device15();
AssertTrue(Condition := device15.outSignal, Message := 'Rejected command cannot change output intent');
TEST_FINISHED();
END_METHOD

METHOD AnalogSetValueRejectsInvalidIdentity
TEST('AnalogSetValueRejectsInvalidIdentity');
device16.SetValue(rValue := 25.0); device16();
rsp := device16.SetValue(rValue := 80.0, eRequester := invalid^);
AssertEquals_DINT(Expected := TcForge.E_RpcMethodResponse.REJECTED_INVALID_PARAMETER, Actual := rsp, Message := 'Invalid identity must reject before device-specific logic');
device16();
AssertEquals_REAL(Expected := 25.0, Actual := device16.sts.commanded, Delta := 0.001, Message := 'Rejected request preserves commanded value');
TEST_FINISHED();
END_METHOD

METHOD AnalogForceSafeRejectsInvalidIdentity
TEST('AnalogForceSafeRejectsInvalidIdentity');
device17.SetValue(rValue := 25.0); device17();
rsp := device17.ForceSafe(eRequester := invalid^);
AssertEquals_DINT(Expected := TcForge.E_RpcMethodResponse.REJECTED_INVALID_PARAMETER, Actual := rsp, Message := 'Invalid identity must reject before device-specific logic');
device17();
AssertEquals_REAL(Expected := 25.0, Actual := device17.sts.commanded, Delta := 0.001, Message := 'Rejected request preserves commanded value');
TEST_FINISHED();
END_METHOD

METHOD AnalogResetRejectsInvalidIdentity
TEST('AnalogResetRejectsInvalidIdentity');
device18.SetValue(rValue := 25.0); device18();
rsp := device18.Reset(eRequester := invalid^);
AssertEquals_DINT(Expected := TcForge.E_RpcMethodResponse.REJECTED_INVALID_PARAMETER, Actual := rsp, Message := 'Invalid identity must reject before device-specific logic');
device18();
AssertEquals_REAL(Expected := 25.0, Actual := device18.sts.commanded, Delta := 0.001, Message := 'Rejected request preserves commanded value');
TEST_FINISHED();
END_METHOD

METHOD BaseResetRejectsInvalidIdentity
TEST('BaseResetRejectsInvalidIdentity');
device19.ProbeRaise(code := 42, source := 'TEST', reason := 'Preserve fault');
rsp := device19.Reset(eRequester := invalid^);
AssertEquals_DINT(Expected := TcForge.E_RpcMethodResponse.REJECTED_INVALID_PARAMETER, Actual := rsp, Message := 'Invalid identity must reject before device-specific logic');
AssertEquals_DINT(Expected := 42, Actual := device19.GetFaultCode(), Message := 'Rejected reset preserves fault');
TEST_FINISHED();
END_METHOD

METHOD AlarmAckRejectsInvalidIdentity
TEST('AlarmAckRejectsInvalidIdentity');

rsp := device20.Ack(eRequester := invalid^);
AssertEquals_DINT(Expected := TcForge.E_RpcMethodResponse.REJECTED_INVALID_PARAMETER, Actual := rsp, Message := 'Invalid identity must reject before device-specific logic');

TEST_FINISHED();
END_METHOD

METHOD LimitAlarmAckRejectsInvalidIdentity
TEST('LimitAlarmAckRejectsInvalidIdentity');

rsp := device21.Ack(eRequester := invalid^);
AssertEquals_DINT(Expected := TcForge.E_RpcMethodResponse.REJECTED_INVALID_PARAMETER, Actual := rsp, Message := 'Invalid identity must reject before device-specific logic');

TEST_FINISHED();
END_METHOD

END_FUNCTION_BLOCK

// ---- Testing/POUs/FB_StateMachine_Probe.TcPOU
// Test-only access to state, timer and permissive internals for isolated cases.
// The cyclic body supplies one synthetic active-step observation before SUPER^()
// because transition unit tests do not run a complete application scan.
// Coverage regressions use real FB_StateMachine instances instead of this probe.
// Plain VAR members are accessible to TwinCAT subclasses. This type is excluded
// from the shipped library.
FUNCTION_BLOCK FB_StateMachine_Probe EXTENDS TcForge.FB_StateMachine

// Transition unit tests supply no full application scan. Coverage is tested with real FB_StateMachine instances.
_activeStepCalls := 1;
SUPER^();

// Full isolation reset for the shared suite-level probe. Clears fault
// book-keeping, command-request flags, permissive / interlock live
// state, rising-edge memory on the SM's internal triggers, and
// published Status back to its power-on values. Each test method
// calls this in its own Setup() so tests see a clean slate even
// though the probe instance itself is reused.
//
METHOD PUBLIC ResetAll
VAR
    i : UDINT;
END_VAR
_ClearFault();
_stepFailurePending := FALSE;
_stepRecoveryPending := FALSE;
_coverageStep := -1;
_activeStepCalls := 0;
Status.ShutdownFailed := FALSE;
Status.FailedStep := 0;
inpShutdownConfirmed := FALSE;
bSourceLockedToProg := FALSE;
Status.AtRecoveryStep := FALSE;
inpSubmoduleFaulted := FALSE;

_abortRequested         := FALSE;
_completeStateRequested := FALSE;
_homeRequested          := FALSE;
_pauseRequested         := FALSE;
_proceedRequested       := FALSE;
_startRequested         := FALSE;
_stopRequested          := FALSE;
_retryActive            := FALSE;
RetryComplete           := FALSE;
_blockedCode            := 0;
_starvedCode            := 0;

// Order matters for FB_Interlock: Reset() snaps _latchedBits to the
// current nLiveBits, so the live bits must already be good before the
// reset. Otherwise a bit left FALSE by a previous test (e.g. the
// running-interlock-trip case) stays latched bad across the reset and
// makes every subsequent test look like the interlock auto-aborted.
// FB_Permissives is non-latching so the order doesn't matter there,
// but we keep it consistent.
FOR i := 0 TO 63 DO
    permHome.MapInput(bitIndex := i, inputValue := TRUE);
    permStart.MapInput(bitIndex := i, inputValue := TRUE);
    permProceed.MapInput(bitIndex := i, inputValue := TRUE);
    permAuto.MapInput(bitIndex := i, inputValue := TRUE);
    intlkRunning.MapInput(bitIndex := i, inputValue := TRUE);
END_FOR;
cfgAutoRun := FALSE;
StepTimer(IN := FALSE);
permHome.Reset();
permStart.Reset();
permProceed.Reset();
permAuto.Reset();
intlkRunning.Reset();

R_TRIG_1(CLK := FALSE);

Status.State            := TcForge.E_SM_State.STOPPED;
Status.LastState        := TcForge.E_SM_State.STOPPED;
Status.Step.Current     := 0;
Status.Step.Next        := 0;
Status.Step.TimerSeconds := 0.0;
Status.Faulted          := FALSE;
Status.SubmoduleFaulted := FALSE;
Status.BlockedCondition := 0;
Status.StarvedCondition := 0;
Status.AutoCycleRequest := FALSE;

_nextStep      := 0;
_returnState   := TcForge.E_SM_State.STOPPED;
ReturnNextStep := 0;
PreviousStep   := 0;
END_METHOD

// Force the active step number. Lets FB_Step see _active = TRUE without
// us having to drive Home/Start/state transitions end-to-end.
METHOD PUBLIC SetCurrentStep
VAR_INPUT
    nStep : DINT;
END_VAR
Status.Step.Current := nStep;
END_METHOD

// Inject a step-timer reading so timeout branches can be tested without
// actually letting wall-clock time pass. The production SM owns the
// timer — here we just write the published value directly.
METHOD PUBLIC SetTimerSeconds
VAR_INPUT
    seconds : REAL;
END_VAR
Status.Step.TimerSeconds := seconds;
END_METHOD

// Park the SM in a specific state without walking the full
// Home/Start/Complete command sequence. Used by the transition tests
// to set up "machine is in state X, now issue command Y" without
// running a sequence first.
METHOD PUBLIC ForceState
VAR_INPUT
    state : TcForge.E_SM_State;
END_VAR
Status.State := state;
END_METHOD

// Set Status.LastState directly. Needed for the AutoCycle path
// (fires when State=READY AND LastState=RUNNING) without walking
// a full RUNNING -> READY transition first.
METHOD PUBLIC ForceLastState
VAR_INPUT
    state : TcForge.E_SM_State;
END_VAR
Status.LastState := state;
END_METHOD

// Drive _nextStep directly. Used with ForceState+SetCurrentStep to
// simulate "mid-sequence" — if _nextStep stays at 0 while a forced
// Current lands inside the state's step range, R_TRIG_5 fires a
// spurious sequence-complete that tests don't want.
METHOD PUBLIC ForceNextStep
VAR_INPUT
    nStep : DINT;
END_VAR
_nextStep := nStep;
END_METHOD

// Map a bit into the private permHome block so the Home-permissive
// gate can be observed. Without this the internal FB_Permissives has
// no external mapping surface on the SM, and every test would see
// "all perms OK" by default.
METHOD PUBLIC MapHomePerm
VAR_INPUT
    bitIndex : UDINT;
    bGood    : BOOL;
END_VAR
permHome.MapInput(bitIndex := bitIndex, inputValue := bGood);
END_METHOD

METHOD PUBLIC MapStartPerm
VAR_INPUT
    bitIndex : UDINT;
    bGood    : BOOL;
END_VAR
permStart.MapInput(bitIndex := bitIndex, inputValue := bGood);
END_METHOD

METHOD PUBLIC MapProceedPerm
VAR_INPUT
    bitIndex : UDINT;
    bGood    : BOOL;
END_VAR
permProceed.MapInput(bitIndex := bitIndex, inputValue := bGood);
END_METHOD

METHOD PUBLIC MapAutoPerm
VAR_INPUT
    bitIndex : UDINT;
    bGood    : BOOL;
END_VAR
permAuto.MapInput(bitIndex := bitIndex, inputValue := bGood);
END_METHOD

END_FUNCTION_BLOCK

// ---- Testing/POUs/FB_DeviceBase_Probe.TcPOU
// Test-only concrete child of FB_DeviceBase. Exposes the protected API
// (_Raise / _ClearFault / _AcceptCommand / _UpdateHeader) through public
// "Probe*" wrappers so FB_DeviceBase_Test can drive the base contract
// without a full device FB in the way. Also overrides ResolveFaultString
// so the tests can verify virtual dispatch.
//
// This FB lives in the Testing project on purpose — it is not part of the
// TcForge public surface.
FUNCTION_BLOCK FB_DeviceBase_Probe EXTENDS TcForge.FB_DeviceBase
VAR_OUTPUT
    header : TcForge.ST_DeviceHeader_Sts;
END_VAR

// Nothing cyclic — tests call the probe methods directly.

METHOD PUBLIC ProbeRaise : BOOL
VAR_INPUT
    code   : DINT;
    source : STRING(31);
    reason : STRING(79);
END_VAR
ProbeRaise := _Raise(code := code, source := source, reason := reason);
END_METHOD

METHOD PUBLIC ProbeClearFault
_ClearFault();
END_METHOD

METHOD PUBLIC ProbeAcceptCommand
VAR_INPUT
    eRequester : TcForge.E_Requester;
END_VAR
_AcceptCommand(eRequester := eRequester);
END_METHOD

// Populate the probe's own header struct via the protected _UpdateHeader.
METHOD PUBLIC Refresh
VAR_INPUT
    stateString : STRING(31);
    busy     : BOOL;
END_VAR
_UpdateHeader(
    header      := header,
    stateString := stateString,
    busy     := busy);
END_METHOD

// Minimal resolver so the tests can verify virtual dispatch through the
// base's GetFaultString() / _UpdateHeader() calls. Maps a few well-known
// codes; everything else returns empty (inherited default behaviour).
METHOD PROTECTED ResolveFaultString : STRING(79)
VAR_INPUT
    code : DINT;
END_VAR
CASE code OF
    42: ResolveFaultString := 'Motion timeout';
    99: ResolveFaultString := 'Limit tripped';
ELSE
    ResolveFaultString := '';
END_CASE;
END_METHOD

END_FUNCTION_BLOCK

// ---- Testing/POUs/FB_RpcContext_Probe.TcPOU
FUNCTION_BLOCK FB_RpcContext_Probe
VAR_OUTPUT ownerTask : DINT; END_VAR

ownerTask := Tc2_System.GETCURTASKINDEXEX();

{attribute 'TcRpcEnable' := '1'}
METHOD PUBLIC ReadContext : DINT
ReadContext := Tc2_System.GETCURTASKINDEXEX();
END_METHOD

END_FUNCTION_BLOCK

// ---- Testing/Tests/FB_AssemblyStation_Test.TcPOU
// Functional tests use deterministic cylinder feedback, not a real IO bus.
// Each scenario owns a station instance and runs in the existing TcUnit task.
FUNCTION_BLOCK FB_AssemblyStation_Test EXTENDS TcUnit.FB_TestSuite
VAR
    machines : ARRAY[0..4] OF FB_AssemblyStation;
    phase : ARRAY[0..4] OF UINT;
    done : ARRAY[0..4] OF BOOL;
    injected : ARRAY[0..4] OF BOOL;
    sawPress : ARRAY[0..4] OF BOOL;
    sawEject : ARRAY[0..4] OF BOOL;
    recoveryPhase : UINT;
    watchdog : ARRAY[0..4] OF TON;
END_VAR

CompleteAssemblyCycle();
QualityLossStopsAllAxes();
LostClampPreventsPressMotion();
BlockedDischargeRejectsEjection();
BadHeightCannotCompleteInspection();

METHOD CompleteAssemblyCycle
IF done[0] THEN
    RETURN;
END_IF;
TEST('CompleteAssemblyCycle');

// Initialize the plant at home with a part ready to assemble.
IF phase[0] = 0 THEN
    machines[0].inputs.clamp.retracted := TRUE;
    machines[0].inputs.press.retracted := TRUE;
    machines[0].inputs.ejector.retracted := TRUE;
    machines[0].inputs.partPresent := TRUE;
    machines[0].inputs.dischargeClear := TRUE;
    machines[0].inputs.pressureRaw := 19660;
    machines[0].inputs.heightRaw := 16384;
    machines[0].inputs.inputQuality := TcForge.E_IO_Quality.GOOD;
    machines[0].inputs.outputQuality := TcForge.E_IO_Quality.GOOD;
    machines[0].inputs.shutdownQuality := TcForge.E_IO_Quality.GOOD;
    machines[0].inputs.shutdownConfirmed := TRUE;
END_IF;

// Move feedback on the following scan, only in response to actual coil outputs.
IF machines[0].outputs.clamp.advance THEN
    machines[0].inputs.clamp.advanced := TRUE;
    machines[0].inputs.clamp.retracted := FALSE;
ELSIF machines[0].outputs.clamp.retract THEN
    machines[0].inputs.clamp.advanced := FALSE;
    machines[0].inputs.clamp.retracted := TRUE;
END_IF;

IF machines[0].outputs.press.advance THEN
    machines[0].inputs.press.advanced := TRUE;
    machines[0].inputs.press.retracted := FALSE;
ELSIF machines[0].outputs.press.retract THEN
    machines[0].inputs.press.advanced := FALSE;
    machines[0].inputs.press.retracted := TRUE;
END_IF;

IF machines[0].outputs.ejector.advance THEN
    machines[0].inputs.ejector.advanced := TRUE;
    machines[0].inputs.ejector.retracted := FALSE;
ELSIF machines[0].outputs.ejector.retract THEN
    machines[0].inputs.ejector.advanced := FALSE;
    machines[0].inputs.ejector.retracted := TRUE;
END_IF;

IF machines[0].outputs.ejector.advance THEN
    machines[0].inputs.partPresent := FALSE;
    sawEject[0] := TRUE;
END_IF;
IF machines[0].outputs.press.advance THEN
    sawPress[0] := TRUE;
END_IF;

machines[0].command := E_ReferenceCommand.None;
CASE phase[0] OF
0:
    phase[0] := 1;
1:
    machines[0].command := E_ReferenceCommand.Home;
    phase[0] := 2;
2:
    IF machines[0].sequence.State = TcForge.E_SM_State.READY THEN
        phase[0] := 3;
    END_IF;
3:
    machines[0].command := E_ReferenceCommand.Start;
    phase[0] := 4;
END_CASE;

machines[0]();

AssertFalse(
    Condition := machines[0].outputs.clamp.advance AND machines[0].outputs.clamp.retract,
    Message := 'clamp: opposing coils must never energize together'
);
AssertFalse(
    Condition := machines[0].outputs.press.advance AND machines[0].outputs.press.retract,
    Message := 'press: opposing coils must never energize together'
);
AssertFalse(
    Condition := machines[0].outputs.ejector.advance AND machines[0].outputs.ejector.retract,
    Message := 'ejector: opposing coils must never energize together'
);
IF phase[0] = 4 AND sawPress[0] AND sawEject[0]
    AND machines[0].sequence.State = TcForge.E_SM_State.READY THEN
    AssertFalse(Condition := machines[0].sequence.Faulted, Message := 'Assembly completes without fault');
    AssertTrue(Condition := machines[0].inputs.ejector.retracted, Message := 'Ejector returns home');
    done[0] := TRUE;
END_IF;

watchdog[0](IN := TRUE, PT := T#18S);
IF watchdog[0].Q AND NOT done[0] THEN
    AssertTrue(Condition := FALSE, Message := 'Assembly scenario timed out');
    done[0] := TRUE;
END_IF;
IF done[0] THEN
    TEST_FINISHED();
END_IF;
END_METHOD

METHOD QualityLossStopsAllAxes
IF done[1] THEN
    RETURN;
END_IF;
TEST('QualityLossStopsAllAxes');

// Initialize the plant at home with a part ready to assemble.
IF phase[1] = 0 THEN
    machines[1].inputs.clamp.retracted := TRUE;
    machines[1].inputs.press.retracted := TRUE;
    machines[1].inputs.ejector.retracted := TRUE;
    machines[1].inputs.partPresent := TRUE;
    machines[1].inputs.dischargeClear := TRUE;
    machines[1].inputs.pressureRaw := 19660;
    machines[1].inputs.heightRaw := 16384;
    machines[1].inputs.inputQuality := TcForge.E_IO_Quality.GOOD;
    machines[1].inputs.outputQuality := TcForge.E_IO_Quality.GOOD;
    machines[1].inputs.shutdownQuality := TcForge.E_IO_Quality.GOOD;
    machines[1].inputs.shutdownConfirmed := TRUE;
END_IF;

// Move feedback on the following scan, only in response to actual coil outputs.
IF machines[1].outputs.clamp.advance THEN
    machines[1].inputs.clamp.advanced := TRUE;
    machines[1].inputs.clamp.retracted := FALSE;
ELSIF machines[1].outputs.clamp.retract THEN
    machines[1].inputs.clamp.advanced := FALSE;
    machines[1].inputs.clamp.retracted := TRUE;
END_IF;

IF machines[1].outputs.press.advance THEN
    machines[1].inputs.press.advanced := TRUE;
    machines[1].inputs.press.retracted := FALSE;
ELSIF machines[1].outputs.press.retract THEN
    machines[1].inputs.press.advanced := FALSE;
    machines[1].inputs.press.retracted := TRUE;
END_IF;

IF machines[1].outputs.ejector.advance THEN
    machines[1].inputs.ejector.advanced := TRUE;
    machines[1].inputs.ejector.retracted := FALSE;
ELSIF machines[1].outputs.ejector.retract THEN
    machines[1].inputs.ejector.advanced := FALSE;
    machines[1].inputs.ejector.retracted := TRUE;
END_IF;

IF machines[1].outputs.ejector.advance THEN
    machines[1].inputs.partPresent := FALSE;
    sawEject[1] := TRUE;
END_IF;
IF machines[1].outputs.press.advance THEN
    sawPress[1] := TRUE;
END_IF;

machines[1].command := E_ReferenceCommand.None;
CASE phase[1] OF
0:
    phase[1] := 1;
1:
    machines[1].command := E_ReferenceCommand.Home;
    phase[1] := 2;
2:
    IF machines[1].sequence.State = TcForge.E_SM_State.READY THEN
        phase[1] := 3;
    END_IF;
3:
    machines[1].command := E_ReferenceCommand.Start;
    phase[1] := 4;
END_CASE;

// Inject this fault only after the relevant machine phase has been reached.
IF sawPress[1] AND recoveryPhase = 0 THEN
    injected[1] := TRUE;
END_IF;
IF injected[1] AND recoveryPhase = 0 THEN
    machines[1].inputs.inputQuality := TcForge.E_IO_Quality.BAD;
END_IF;

IF recoveryPhase = 1 THEN
    machines[1].inputs.inputQuality := TcForge.E_IO_Quality.GOOD;
    IF machines[1].sequence.State = TcForge.E_SM_State.STOPPED THEN
        machines[1].command := E_ReferenceCommand.Reset;
        recoveryPhase := 2;
    END_IF;
ELSIF recoveryPhase = 2 THEN
    machines[1].command := E_ReferenceCommand.None;
END_IF;

machines[1]();

AssertFalse(
    Condition := machines[1].outputs.clamp.advance AND machines[1].outputs.clamp.retract,
    Message := 'clamp: opposing coils must never energize together'
);
AssertFalse(
    Condition := machines[1].outputs.press.advance AND machines[1].outputs.press.retract,
    Message := 'press: opposing coils must never energize together'
);
AssertFalse(
    Condition := machines[1].outputs.ejector.advance AND machines[1].outputs.ejector.retract,
    Message := 'ejector: opposing coils must never energize together'
);
IF injected[1] AND recoveryPhase = 0 THEN
    AssertTrue(Condition := machines[1].outputsInhibited, Message := 'Fault inhibits same scan');
    AssertFalse(
        Condition := machines[1].outputs.press.advance OR machines[1].outputs.clamp.advance
            OR machines[1].outputs.ejector.advance,
        Message := 'No advance output survives invalid evidence'
    );
    recoveryPhase := 1;
ELSIF recoveryPhase = 2 THEN
    AssertEquals_DINT(
        Expected := TcForge.E_RpcMethodResponse.ACCEPTED,
        Actual := machines[1].lastResponse,
        Message := 'One stationary Reset clears recovered device and parent faults'
    );
    AssertTrue(Condition := machines[1].outputsInhibited, Message := 'Reset does not restart motion');
    done[1] := TRUE;
END_IF;

watchdog[1](IN := TRUE, PT := T#18S);
IF watchdog[1].Q AND NOT done[1] THEN
    AssertTrue(Condition := FALSE, Message := 'Assembly scenario timed out');
    done[1] := TRUE;
END_IF;
IF done[1] THEN
    TEST_FINISHED();
END_IF;
END_METHOD

METHOD LostClampPreventsPressMotion
IF done[2] THEN
    RETURN;
END_IF;
TEST('LostClampPreventsPressMotion');

// Initialize the plant at home with a part ready to assemble.
IF phase[2] = 0 THEN
    machines[2].inputs.clamp.retracted := TRUE;
    machines[2].inputs.press.retracted := TRUE;
    machines[2].inputs.ejector.retracted := TRUE;
    machines[2].inputs.partPresent := TRUE;
    machines[2].inputs.dischargeClear := TRUE;
    machines[2].inputs.pressureRaw := 19660;
    machines[2].inputs.heightRaw := 16384;
    machines[2].inputs.inputQuality := TcForge.E_IO_Quality.GOOD;
    machines[2].inputs.outputQuality := TcForge.E_IO_Quality.GOOD;
    machines[2].inputs.shutdownQuality := TcForge.E_IO_Quality.GOOD;
    machines[2].inputs.shutdownConfirmed := TRUE;
END_IF;

// Move feedback on the following scan, only in response to actual coil outputs.
IF machines[2].outputs.clamp.advance THEN
    machines[2].inputs.clamp.advanced := TRUE;
    machines[2].inputs.clamp.retracted := FALSE;
ELSIF machines[2].outputs.clamp.retract THEN
    machines[2].inputs.clamp.advanced := FALSE;
    machines[2].inputs.clamp.retracted := TRUE;
END_IF;

IF machines[2].outputs.press.advance THEN
    machines[2].inputs.press.advanced := TRUE;
    machines[2].inputs.press.retracted := FALSE;
ELSIF machines[2].outputs.press.retract THEN
    machines[2].inputs.press.advanced := FALSE;
    machines[2].inputs.press.retracted := TRUE;
END_IF;

IF machines[2].outputs.ejector.advance THEN
    machines[2].inputs.ejector.advanced := TRUE;
    machines[2].inputs.ejector.retracted := FALSE;
ELSIF machines[2].outputs.ejector.retract THEN
    machines[2].inputs.ejector.advanced := FALSE;
    machines[2].inputs.ejector.retracted := TRUE;
END_IF;

IF machines[2].outputs.ejector.advance THEN
    machines[2].inputs.partPresent := FALSE;
    sawEject[2] := TRUE;
END_IF;
IF machines[2].outputs.press.advance THEN
    sawPress[2] := TRUE;
END_IF;

machines[2].command := E_ReferenceCommand.None;
CASE phase[2] OF
0:
    phase[2] := 1;
1:
    machines[2].command := E_ReferenceCommand.Home;
    phase[2] := 2;
2:
    IF machines[2].sequence.State = TcForge.E_SM_State.READY THEN
        phase[2] := 3;
    END_IF;
3:
    machines[2].command := E_ReferenceCommand.Start;
    phase[2] := 4;
END_CASE;

// Inject this fault only after the relevant machine phase has been reached.
IF sawPress[2] THEN
    injected[2] := TRUE;
END_IF;
IF injected[2] THEN
    machines[2].inputs.clamp.advanced := FALSE;
END_IF;

machines[2]();

AssertFalse(
    Condition := machines[2].outputs.clamp.advance AND machines[2].outputs.clamp.retract,
    Message := 'clamp: opposing coils must never energize together'
);
AssertFalse(
    Condition := machines[2].outputs.press.advance AND machines[2].outputs.press.retract,
    Message := 'press: opposing coils must never energize together'
);
AssertFalse(
    Condition := machines[2].outputs.ejector.advance AND machines[2].outputs.ejector.retract,
    Message := 'ejector: opposing coils must never energize together'
);
IF injected[2] THEN
    AssertTrue(Condition := machines[2].outputsInhibited, Message := 'Fault inhibits same scan');
    AssertFalse(
        Condition := machines[2].outputs.press.advance OR machines[2].outputs.clamp.advance
            OR machines[2].outputs.ejector.advance,
        Message := 'No advance output survives invalid evidence'
    );
    done[2] := TRUE;
END_IF;

watchdog[2](IN := TRUE, PT := T#18S);
IF watchdog[2].Q AND NOT done[2] THEN
    AssertTrue(Condition := FALSE, Message := 'Assembly scenario timed out');
    done[2] := TRUE;
END_IF;
IF done[2] THEN
    TEST_FINISHED();
END_IF;
END_METHOD

METHOD BlockedDischargeRejectsEjection
IF done[3] THEN
    RETURN;
END_IF;
TEST('BlockedDischargeRejectsEjection');

// Initialize the plant at home with a part ready to assemble.
IF phase[3] = 0 THEN
    machines[3].inputs.clamp.retracted := TRUE;
    machines[3].inputs.press.retracted := TRUE;
    machines[3].inputs.ejector.retracted := TRUE;
    machines[3].inputs.partPresent := TRUE;
    machines[3].inputs.dischargeClear := TRUE;
    machines[3].inputs.pressureRaw := 19660;
    machines[3].inputs.heightRaw := 16384;
    machines[3].inputs.inputQuality := TcForge.E_IO_Quality.GOOD;
    machines[3].inputs.outputQuality := TcForge.E_IO_Quality.GOOD;
    machines[3].inputs.shutdownQuality := TcForge.E_IO_Quality.GOOD;
    machines[3].inputs.shutdownConfirmed := TRUE;
END_IF;

// Move feedback on the following scan, only in response to actual coil outputs.
IF machines[3].outputs.clamp.advance THEN
    machines[3].inputs.clamp.advanced := TRUE;
    machines[3].inputs.clamp.retracted := FALSE;
ELSIF machines[3].outputs.clamp.retract THEN
    machines[3].inputs.clamp.advanced := FALSE;
    machines[3].inputs.clamp.retracted := TRUE;
END_IF;

IF machines[3].outputs.press.advance THEN
    machines[3].inputs.press.advanced := TRUE;
    machines[3].inputs.press.retracted := FALSE;
ELSIF machines[3].outputs.press.retract THEN
    machines[3].inputs.press.advanced := FALSE;
    machines[3].inputs.press.retracted := TRUE;
END_IF;

IF machines[3].outputs.ejector.advance THEN
    machines[3].inputs.ejector.advanced := TRUE;
    machines[3].inputs.ejector.retracted := FALSE;
ELSIF machines[3].outputs.ejector.retract THEN
    machines[3].inputs.ejector.advanced := FALSE;
    machines[3].inputs.ejector.retracted := TRUE;
END_IF;

IF machines[3].outputs.ejector.advance THEN
    machines[3].inputs.partPresent := FALSE;
    sawEject[3] := TRUE;
END_IF;
IF machines[3].outputs.press.advance THEN
    sawPress[3] := TRUE;
END_IF;

machines[3].command := E_ReferenceCommand.None;
CASE phase[3] OF
0:
    phase[3] := 1;
1:
    machines[3].command := E_ReferenceCommand.Home;
    phase[3] := 2;
2:
    IF machines[3].sequence.State = TcForge.E_SM_State.READY THEN
        phase[3] := 3;
    END_IF;
3:
    machines[3].command := E_ReferenceCommand.Start;
    phase[3] := 4;
END_CASE;

// Inject this fault only after the relevant machine phase has been reached.
IF machines[3].sequence.Step.Current = 3010 THEN
    injected[3] := TRUE;
END_IF;
IF injected[3] THEN
    machines[3].inputs.dischargeClear := FALSE;
END_IF;

machines[3]();

AssertFalse(
    Condition := machines[3].outputs.clamp.advance AND machines[3].outputs.clamp.retract,
    Message := 'clamp: opposing coils must never energize together'
);
AssertFalse(
    Condition := machines[3].outputs.press.advance AND machines[3].outputs.press.retract,
    Message := 'press: opposing coils must never energize together'
);
AssertFalse(
    Condition := machines[3].outputs.ejector.advance AND machines[3].outputs.ejector.retract,
    Message := 'ejector: opposing coils must never energize together'
);
IF injected[3] THEN
    AssertFalse(Condition := machines[3].outputs.ejector.advance, Message := 'Blocked exit cannot eject');
    IF machines[3].sequence.State = TcForge.E_SM_State.ABORTING
        OR machines[3].sequence.State = TcForge.E_SM_State.STOPPED THEN
        done[3] := TRUE;
    END_IF;
END_IF;

watchdog[3](IN := TRUE, PT := T#18S);
IF watchdog[3].Q AND NOT done[3] THEN
    AssertTrue(Condition := FALSE, Message := 'Assembly scenario timed out');
    done[3] := TRUE;
END_IF;
IF done[3] THEN
    TEST_FINISHED();
END_IF;
END_METHOD

METHOD BadHeightCannotCompleteInspection
IF done[4] THEN
    RETURN;
END_IF;
TEST('BadHeightCannotCompleteInspection');

// Initialize the plant at home with a part ready to assemble.
IF phase[4] = 0 THEN
    machines[4].inputs.clamp.retracted := TRUE;
    machines[4].inputs.press.retracted := TRUE;
    machines[4].inputs.ejector.retracted := TRUE;
    machines[4].inputs.partPresent := TRUE;
    machines[4].inputs.dischargeClear := TRUE;
    machines[4].inputs.pressureRaw := 19660;
    machines[4].inputs.heightRaw := 16384;
    machines[4].inputs.inputQuality := TcForge.E_IO_Quality.GOOD;
    machines[4].inputs.outputQuality := TcForge.E_IO_Quality.GOOD;
    machines[4].inputs.shutdownQuality := TcForge.E_IO_Quality.GOOD;
    machines[4].inputs.shutdownConfirmed := TRUE;
END_IF;

// Move feedback on the following scan, only in response to actual coil outputs.
IF machines[4].outputs.clamp.advance THEN
    machines[4].inputs.clamp.advanced := TRUE;
    machines[4].inputs.clamp.retracted := FALSE;
ELSIF machines[4].outputs.clamp.retract THEN
    machines[4].inputs.clamp.advanced := FALSE;
    machines[4].inputs.clamp.retracted := TRUE;
END_IF;

IF machines[4].outputs.press.advance THEN
    machines[4].inputs.press.advanced := TRUE;
    machines[4].inputs.press.retracted := FALSE;
ELSIF machines[4].outputs.press.retract THEN
    machines[4].inputs.press.advanced := FALSE;
    machines[4].inputs.press.retracted := TRUE;
END_IF;

IF machines[4].outputs.ejector.advance THEN
    machines[4].inputs.ejector.advanced := TRUE;
    machines[4].inputs.ejector.retracted := FALSE;
ELSIF machines[4].outputs.ejector.retract THEN
    machines[4].inputs.ejector.advanced := FALSE;
    machines[4].inputs.ejector.retracted := TRUE;
END_IF;

IF machines[4].outputs.ejector.advance THEN
    machines[4].inputs.partPresent := FALSE;
    sawEject[4] := TRUE;
END_IF;
IF machines[4].outputs.press.advance THEN
    sawPress[4] := TRUE;
END_IF;

machines[4].command := E_ReferenceCommand.None;
CASE phase[4] OF
0:
    phase[4] := 1;
1:
    machines[4].command := E_ReferenceCommand.Home;
    phase[4] := 2;
2:
    IF machines[4].sequence.State = TcForge.E_SM_State.READY THEN
        phase[4] := 3;
    END_IF;
3:
    machines[4].command := E_ReferenceCommand.Start;
    phase[4] := 4;
END_CASE;

// Inject this fault only after the relevant machine phase has been reached.
IF machines[4].sequence.Step.Current = 3004 THEN
    injected[4] := TRUE;
END_IF;
IF injected[4] THEN
    machines[4].inputs.heightRaw := 1000;
END_IF;

machines[4]();

AssertFalse(
    Condition := machines[4].outputs.clamp.advance AND machines[4].outputs.clamp.retract,
    Message := 'clamp: opposing coils must never energize together'
);
AssertFalse(
    Condition := machines[4].outputs.press.advance AND machines[4].outputs.press.retract,
    Message := 'press: opposing coils must never energize together'
);
AssertFalse(
    Condition := machines[4].outputs.ejector.advance AND machines[4].outputs.ejector.retract,
    Message := 'ejector: opposing coils must never energize together'
);
IF injected[4] THEN
    AssertFalse(Condition := sawEject[4], Message := 'Failed inspection cannot eject');
    IF machines[4].sequence.Faulted THEN
        AssertEquals_DINT(
            Expected := 3006,
            Actual := machines[4].sequence.FailedStep,
            Message := 'Bad height faults the inspection phase'
        );
        done[4] := TRUE;
    END_IF;
END_IF;

watchdog[4](IN := TRUE, PT := T#18S);
IF watchdog[4].Q AND NOT done[4] THEN
    AssertTrue(Condition := FALSE, Message := 'Assembly scenario timed out');
    done[4] := TRUE;
END_IF;
IF done[4] THEN
    TEST_FINISHED();
END_IF;
END_METHOD

END_FUNCTION_BLOCK

// ---- Testing/Tests/FB_ReferenceMachine_Test.TcPOU
FUNCTION_BLOCK FB_ReferenceMachine_Test EXTENDS TcUnit.FB_TestSuite
VAR
    case0_m : FB_ReferenceMachine;
    case0_phase, case0_age : UINT;
    case0_done, case0_seenAdvance, case0_seenRetract : BOOL;
    case0_watchdog : TON;
    case1_m : FB_ReferenceMachine;
    case1_phase, case1_age : UINT;
    case1_done, case1_seenAdvance, case1_seenRetract : BOOL;
    case1_watchdog : TON;
    case2_m : FB_ReferenceMachine;
    case2_phase, case2_age : UINT;
    case2_done, case2_seenAdvance, case2_seenRetract : BOOL;
    case2_watchdog : TON;
    case3_m : FB_ReferenceMachine;
    case3_phase, case3_age : UINT;
    case3_done, case3_seenAdvance, case3_seenRetract : BOOL;
    case3_watchdog : TON;
    case4_m : FB_ReferenceMachine;
    case4_phase, case4_age : UINT;
    case4_done, case4_seenAdvance, case4_seenRetract : BOOL;
    case4_watchdog : TON;
    case5_m : FB_ReferenceMachine;
    case5_phase, case5_age : UINT;
    case5_done, case5_seenAdvance, case5_seenRetract : BOOL;
    case5_watchdog : TON;
    case6_m : FB_ReferenceMachine;
    case6_phase, case6_age : UINT;
    case6_done, case6_seenAdvance, case6_seenRetract : BOOL;
    case6_watchdog : TON;
    case7_m : FB_ReferenceMachine;
    case7_phase, case7_age : UINT;
    case7_done, case7_seenAdvance, case7_seenRetract : BOOL;
    case7_watchdog : TON;
    case8_m : FB_ReferenceMachine;
    case8_phase, case8_age : UINT;
    case8_done, case8_seenAdvance, case8_seenRetract : BOOL;
    case8_watchdog : TON;
    case9_m : FB_ReferenceMachine;
    case9_phase, case9_age : UINT;
    case9_done, case9_seenAdvance, case9_seenRetract : BOOL;
    case9_watchdog : TON;
END_VAR

OutputQualityLossRequiresExplicitRecovery();
AbortRequiresTrustedFeedback();
ResetRejectedDuringMotion();
StartupUnknownInhibits();
HomeAndRunThroughPhysicalBoundary();
ControlledStopCancelsBeforeRetract();
AbortWaitsForIndependentFeedback();
QualityLossRequiresExplicitRecovery();
ContradictoryFeedbackInhibitsSameScan();
AbortTimeoutRequiresConfirmedReset();

METHOD StartupUnknownInhibits
IF case0_done THEN RETURN; END_IF;
TEST('StartupUnknownInhibits');
case0_m();
AssertFalse(Condition := case0_m.outAdvance OR case0_m.outRetract, Message := 'Unknown startup quality inhibits both outputs');
AssertTrue(Condition := case0_m.outputsInhibited, Message := 'Startup inhibition is visible');
case0_done := TRUE;
IF case0_done THEN TEST_FINISHED(); END_IF;
END_METHOD

METHOD HomeAndRunThroughPhysicalBoundary
IF case1_done THEN RETURN; END_IF;
TEST('HomeAndRunThroughPhysicalBoundary');
case1_age := case1_age + 1;
case1_m.command := E_ReferenceCommand.None;
IF case1_phase < 3 THEN
    case1_m.inputQuality := TcForge.E_IO_Quality.GOOD; case1_m.outputQuality := TcForge.E_IO_Quality.GOOD;
    case1_m.shutdownQuality := TcForge.E_IO_Quality.GOOD; case1_m.shutdownConfirmed := TRUE; case1_m.inRetracted := TRUE;
    CASE case1_phase OF
    0: case1_phase := 1;
    1: case1_m.command := E_ReferenceCommand.Home; case1_phase := 2;
    2: IF case1_m.sequence.State = TcForge.E_SM_State.READY THEN case1_phase := 3; END_IF;
    END_CASE;
ELSE
CASE case1_phase OF
3:
    case1_m.command := E_ReferenceCommand.Start; case1_phase := 4;
4:
    // Hold Start: completing the cycle must not start another one.
    case1_m.command := E_ReferenceCommand.Start;
    IF case1_m.outAdvance THEN case1_m.inAdvanced := TRUE; case1_m.inRetracted := FALSE; case1_seenAdvance := TRUE; END_IF;
    IF case1_m.outRetract THEN case1_m.inRetracted := TRUE; case1_m.inAdvanced := FALSE; case1_seenRetract := TRUE; END_IF;
    IF case1_seenAdvance AND case1_m.sequence.State = TcForge.E_SM_State.READY THEN case1_phase := 5; END_IF;
5:
    case1_m.command := E_ReferenceCommand.Start;
    IF case1_age > 50 THEN
        AssertTrue(Condition := case1_seenAdvance AND case1_seenRetract, Message := 'Both real output paths exercised');
        AssertEquals_DINT(Expected := TcForge.E_SM_State.READY, Actual := case1_m.sequence.State, Message := 'Held Start cannot retrigger');
        case1_done := TRUE;
    END_IF;
END_CASE;
END_IF;
case1_m();
AssertFalse(Condition := case1_m.outAdvance AND case1_m.outRetract, Message := 'Coils must remain mutually exclusive');
case1_watchdog(IN := TRUE, PT := T#8S);
IF case1_watchdog.Q AND NOT case1_done THEN AssertTrue(Condition := FALSE, Message := 'Scenario did not reach its expected state'); case1_done := TRUE; END_IF;
IF case1_done THEN TEST_FINISHED(); END_IF;
END_METHOD

METHOD ControlledStopCancelsBeforeRetract
IF case2_done THEN RETURN; END_IF;
TEST('ControlledStopCancelsBeforeRetract');
case2_age := case2_age + 1;
case2_m.command := E_ReferenceCommand.None;
IF case2_phase < 3 THEN
    case2_m.inputQuality := TcForge.E_IO_Quality.GOOD; case2_m.outputQuality := TcForge.E_IO_Quality.GOOD;
    case2_m.shutdownQuality := TcForge.E_IO_Quality.GOOD; case2_m.shutdownConfirmed := TRUE; case2_m.inRetracted := TRUE;
    CASE case2_phase OF
    0: case2_phase := 1;
    1: case2_m.command := E_ReferenceCommand.Home; case2_phase := 2;
    2: IF case2_m.sequence.State = TcForge.E_SM_State.READY THEN case2_phase := 3; END_IF;
    END_CASE;
ELSE
CASE case2_phase OF
3: case2_m.command := E_ReferenceCommand.Start; case2_phase := 4;
4:
    IF case2_m.outAdvance THEN case2_m.inRetracted := FALSE; case2_m.command := E_ReferenceCommand.Stop; case2_phase := 5; END_IF;
5:
    AssertFalse(Condition := case2_m.outAdvance, Message := 'Stop cancels advance before retracting');
    IF case2_m.outRetract THEN case2_seenRetract := TRUE; case2_m.inRetracted := TRUE; END_IF;
    IF case2_m.sequence.State = TcForge.E_SM_State.STOPPED THEN
        AssertTrue(Condition := case2_seenRetract, Message := 'Controlled Stop physically retracts');
        AssertFalse(Condition := case2_m.faulted OR case2_m.outAdvance OR case2_m.outRetract, Message := 'Healthy Stop finishes inhibited');
        case2_done := TRUE;
    END_IF;
END_CASE;
END_IF;
case2_m();
AssertFalse(Condition := case2_m.outAdvance AND case2_m.outRetract, Message := 'Coils must remain mutually exclusive');
case2_watchdog(IN := TRUE, PT := T#8S);
IF case2_watchdog.Q AND NOT case2_done THEN AssertTrue(Condition := FALSE, Message := 'Scenario did not reach its expected state'); case2_done := TRUE; END_IF;
IF case2_done THEN TEST_FINISHED(); END_IF;
END_METHOD

METHOD AbortWaitsForIndependentFeedback
IF case3_done THEN RETURN; END_IF;
TEST('AbortWaitsForIndependentFeedback');
case3_age := case3_age + 1;
case3_m.command := E_ReferenceCommand.None;
IF case3_phase < 3 THEN
    case3_m.inputQuality := TcForge.E_IO_Quality.GOOD; case3_m.outputQuality := TcForge.E_IO_Quality.GOOD;
    case3_m.shutdownQuality := TcForge.E_IO_Quality.GOOD; case3_m.shutdownConfirmed := TRUE; case3_m.inRetracted := TRUE;
    CASE case3_phase OF
    0: case3_phase := 1;
    1: case3_m.command := E_ReferenceCommand.Home; case3_phase := 2;
    2: IF case3_m.sequence.State = TcForge.E_SM_State.READY THEN case3_phase := 3; END_IF;
    END_CASE;
ELSE
CASE case3_phase OF
3: case3_m.command := E_ReferenceCommand.Start; case3_phase := 4;
4:
    IF case3_m.outAdvance THEN case3_m.shutdownConfirmed := FALSE; case3_m.command := E_ReferenceCommand.Abort; case3_phase := 5; END_IF;
5:
    AssertFalse(Condition := case3_m.outAdvance OR case3_m.outRetract, Message := 'Abort removes both coils');
    IF case3_age > 35 THEN
        AssertEquals_DINT(Expected := TcForge.E_SM_State.ABORTING, Actual := case3_m.sequence.State, Message := 'Coil commands do not confirm shutdown');
        case3_m.shutdownConfirmed := TRUE; case3_phase := 6;
    END_IF;
6:
    IF case3_m.sequence.State = TcForge.E_SM_State.STOPPED THEN case3_done := TRUE; END_IF;
END_CASE;
END_IF;
case3_m();
AssertFalse(Condition := case3_m.outAdvance AND case3_m.outRetract, Message := 'Coils must remain mutually exclusive');
case3_watchdog(IN := TRUE, PT := T#8S);
IF case3_watchdog.Q AND NOT case3_done THEN AssertTrue(Condition := FALSE, Message := 'Scenario did not reach its expected state'); case3_done := TRUE; END_IF;
IF case3_done THEN TEST_FINISHED(); END_IF;
END_METHOD

METHOD QualityLossRequiresExplicitRecovery
IF case4_done THEN RETURN; END_IF;
TEST('QualityLossRequiresExplicitRecovery');
case4_age := case4_age + 1;
case4_m.command := E_ReferenceCommand.None;
IF case4_phase < 3 THEN
    case4_m.inputQuality := TcForge.E_IO_Quality.GOOD; case4_m.outputQuality := TcForge.E_IO_Quality.GOOD;
    case4_m.shutdownQuality := TcForge.E_IO_Quality.GOOD; case4_m.shutdownConfirmed := TRUE; case4_m.inRetracted := TRUE;
    CASE case4_phase OF
    0: case4_phase := 1;
    1: case4_m.command := E_ReferenceCommand.Home; case4_phase := 2;
    2: IF case4_m.sequence.State = TcForge.E_SM_State.READY THEN case4_phase := 3; END_IF;
    END_CASE;
ELSE
CASE case4_phase OF
3: case4_m.command := E_ReferenceCommand.Start; case4_phase := 4;
4:
    IF case4_m.outAdvance THEN case4_m.inputQuality := TcForge.E_IO_Quality.BAD; case4_phase := 5; END_IF;
5:
    AssertFalse(Condition := case4_m.outAdvance OR case4_m.outRetract, Message := 'Quality loss removes outputs in detecting scan');
    IF case4_m.sequence.State = TcForge.E_SM_State.STOPPED THEN case4_m.inputQuality := TcForge.E_IO_Quality.GOOD; case4_phase := 6; END_IF;
6:
    AssertFalse(Condition := case4_m.outAdvance OR case4_m.outRetract, Message := 'Quality restoration cannot restore motion');
    case4_m.command := E_ReferenceCommand.Home; case4_phase := 7;
7:
    AssertTrue(Condition := case4_m.lastResponse <> TcForge.E_RpcMethodResponse.ACCEPTED, Message := 'Home rejected before recovery');
    case4_m.command := E_ReferenceCommand.Reset; case4_phase := 8;
8:
    AssertEquals_DINT(Expected := TcForge.E_RpcMethodResponse.ACCEPTED, Actual := case4_m.lastResponse, Message := 'Healthy confirmed reset accepted');
    AssertFalse(Condition := case4_m.outAdvance OR case4_m.outRetract, Message := 'Reset does not energize outputs');
    case4_phase := 9;
9: case4_m.command := E_ReferenceCommand.Home; case4_phase := 10;
10:
    IF case4_m.sequence.State = TcForge.E_SM_State.READY THEN
        AssertFalse(Condition := case4_m.faulted, Message := 'Explicit recovery permits new Home');
        case4_done := TRUE;
    END_IF;
END_CASE;
END_IF;
case4_m();
AssertFalse(Condition := case4_m.outAdvance AND case4_m.outRetract, Message := 'Coils must remain mutually exclusive');
case4_watchdog(IN := TRUE, PT := T#8S);
IF case4_watchdog.Q AND NOT case4_done THEN AssertTrue(Condition := FALSE, Message := 'Scenario did not reach its expected state'); case4_done := TRUE; END_IF;
IF case4_done THEN TEST_FINISHED(); END_IF;
END_METHOD

METHOD ContradictoryFeedbackInhibitsSameScan
IF case5_done THEN RETURN; END_IF;
TEST('ContradictoryFeedbackInhibitsSameScan');
case5_age := case5_age + 1;
case5_m.command := E_ReferenceCommand.None;
IF case5_phase < 3 THEN
    case5_m.inputQuality := TcForge.E_IO_Quality.GOOD; case5_m.outputQuality := TcForge.E_IO_Quality.GOOD;
    case5_m.shutdownQuality := TcForge.E_IO_Quality.GOOD; case5_m.shutdownConfirmed := TRUE; case5_m.inRetracted := TRUE;
    CASE case5_phase OF
    0: case5_phase := 1;
    1: case5_m.command := E_ReferenceCommand.Home; case5_phase := 2;
    2: IF case5_m.sequence.State = TcForge.E_SM_State.READY THEN case5_phase := 3; END_IF;
    END_CASE;
ELSE
CASE case5_phase OF
3: case5_m.command := E_ReferenceCommand.Start; case5_phase := 4;
4:
    IF case5_m.outAdvance THEN case5_m.inAdvanced := TRUE; case5_m.inRetracted := TRUE; case5_phase := 5; END_IF;
5:
    AssertFalse(Condition := case5_m.outAdvance OR case5_m.outRetract, Message := 'Contradictory feedback removes final outputs same scan');
    AssertTrue(Condition := case5_m.faulted, Message := 'Aggregate status includes fresh actuator fault');
    case5_done := TRUE;
END_CASE;
END_IF;
case5_m();
AssertFalse(Condition := case5_m.outAdvance AND case5_m.outRetract, Message := 'Coils must remain mutually exclusive');
case5_watchdog(IN := TRUE, PT := T#8S);
IF case5_watchdog.Q AND NOT case5_done THEN AssertTrue(Condition := FALSE, Message := 'Scenario did not reach its expected state'); case5_done := TRUE; END_IF;
IF case5_done THEN TEST_FINISHED(); END_IF;
END_METHOD

METHOD AbortTimeoutRequiresConfirmedReset
IF case6_done THEN RETURN; END_IF;
TEST('AbortTimeoutRequiresConfirmedReset');
case6_age := case6_age + 1;
case6_m.command := E_ReferenceCommand.None;
IF case6_phase < 3 THEN
    case6_m.inputQuality := TcForge.E_IO_Quality.GOOD; case6_m.outputQuality := TcForge.E_IO_Quality.GOOD;
    case6_m.shutdownQuality := TcForge.E_IO_Quality.GOOD; case6_m.shutdownConfirmed := TRUE; case6_m.inRetracted := TRUE;
    CASE case6_phase OF
    0: case6_phase := 1;
    1: case6_m.command := E_ReferenceCommand.Home; case6_phase := 2;
    2: IF case6_m.sequence.State = TcForge.E_SM_State.READY THEN case6_phase := 3; END_IF;
    END_CASE;
ELSE
CASE case6_phase OF
3: case6_m.command := E_ReferenceCommand.Abort; case6_m.shutdownConfirmed := FALSE; case6_phase := 4;
4:
    IF case6_m.sequence.ShutdownFailed THEN case6_phase := 5; END_IF;
5:
    IF case6_m.sequence.State = TcForge.E_SM_State.STOPPED THEN case6_m.command := E_ReferenceCommand.Reset; case6_phase := 6; END_IF;
6:
    AssertEquals_DINT(Expected := TcForge.E_RpcMethodResponse.REJECTED_INTERLOCKED, Actual := case6_m.lastResponse, Message := 'Failed Abort cannot reset without feedback');
    AssertTrue(Condition := case6_m.sequence.ShutdownFailed, Message := 'Rejected Reset preserves shutdown failure');
    case6_m.shutdownConfirmed := TRUE; case6_phase := 7;
7: case6_m.command := E_ReferenceCommand.Reset; case6_phase := 8;
8:
    AssertEquals_DINT(Expected := TcForge.E_RpcMethodResponse.ACCEPTED, Actual := case6_m.lastResponse, Message := 'Independent feedback permits Reset');
    AssertFalse(Condition := case6_m.faulted OR case6_m.sequence.ShutdownFailed OR case6_m.outAdvance OR case6_m.outRetract, Message := 'Recovered machine stays deenergized');
    case6_done := TRUE;
END_CASE;
END_IF;
case6_m();
AssertFalse(Condition := case6_m.outAdvance AND case6_m.outRetract, Message := 'Coils must remain mutually exclusive');
case6_watchdog(IN := TRUE, PT := T#8S);
IF case6_watchdog.Q AND NOT case6_done THEN AssertTrue(Condition := FALSE, Message := 'Scenario did not reach its expected state'); case6_done := TRUE; END_IF;
IF case6_done THEN TEST_FINISHED(); END_IF;
END_METHOD

METHOD OutputQualityLossRequiresExplicitRecovery
IF case7_done THEN RETURN; END_IF;
TEST('OutputQualityLossRequiresExplicitRecovery');
case7_age := case7_age + 1;
case7_m.command := E_ReferenceCommand.None;
IF case7_phase < 3 THEN
    case7_m.inputQuality := TcForge.E_IO_Quality.GOOD; case7_m.outputQuality := TcForge.E_IO_Quality.GOOD;
    case7_m.shutdownQuality := TcForge.E_IO_Quality.GOOD; case7_m.shutdownConfirmed := TRUE; case7_m.inRetracted := TRUE;
    CASE case7_phase OF
    0: case7_phase := 1;
    1: case7_m.command := E_ReferenceCommand.Home; case7_phase := 2;
    2: IF case7_m.sequence.State = TcForge.E_SM_State.READY THEN case7_phase := 3; END_IF;
    END_CASE;
ELSE
CASE case7_phase OF
3: case7_m.command := E_ReferenceCommand.Start; case7_phase := 4;
4:
    IF case7_m.outAdvance THEN case7_m.outputQuality := TcForge.E_IO_Quality.BAD; case7_phase := 5; END_IF;
5:
    AssertFalse(Condition := case7_m.outAdvance OR case7_m.outRetract, Message := 'Quality loss removes outputs in detecting scan');
    IF case7_m.sequence.State = TcForge.E_SM_State.STOPPED THEN case7_m.outputQuality := TcForge.E_IO_Quality.GOOD; case7_phase := 6; END_IF;
6:
    AssertFalse(Condition := case7_m.outAdvance OR case7_m.outRetract, Message := 'Quality restoration cannot restore motion');
    case7_m.command := E_ReferenceCommand.Home; case7_phase := 7;
7:
    AssertTrue(Condition := case7_m.lastResponse <> TcForge.E_RpcMethodResponse.ACCEPTED, Message := 'Home rejected before recovery');
    case7_m.command := E_ReferenceCommand.Reset; case7_phase := 8;
8:
    AssertEquals_DINT(Expected := TcForge.E_RpcMethodResponse.ACCEPTED, Actual := case7_m.lastResponse, Message := 'Healthy confirmed reset accepted');
    AssertFalse(Condition := case7_m.outAdvance OR case7_m.outRetract, Message := 'Reset does not energize outputs');
    case7_phase := 9;
9: case7_m.command := E_ReferenceCommand.Home; case7_phase := 10;
10:
    IF case7_m.sequence.State = TcForge.E_SM_State.READY THEN
        AssertFalse(Condition := case7_m.faulted, Message := 'Explicit recovery permits new Home');
        case7_done := TRUE;
    END_IF;
END_CASE;
END_IF;
case7_m();
AssertFalse(Condition := case7_m.outAdvance AND case7_m.outRetract, Message := 'Coils must remain mutually exclusive');
case7_watchdog(IN := TRUE, PT := T#8S);
IF case7_watchdog.Q AND NOT case7_done THEN AssertTrue(Condition := FALSE, Message := 'Scenario did not reach its expected state'); case7_done := TRUE; END_IF;
IF case7_done THEN TEST_FINISHED(); END_IF;
END_METHOD

METHOD AbortRequiresTrustedFeedback
IF case8_done THEN RETURN; END_IF;
TEST('AbortRequiresTrustedFeedback');
case8_age := case8_age + 1;
case8_m.command := E_ReferenceCommand.None;
IF case8_phase < 3 THEN
    case8_m.inputQuality := TcForge.E_IO_Quality.GOOD; case8_m.outputQuality := TcForge.E_IO_Quality.GOOD;
    case8_m.shutdownQuality := TcForge.E_IO_Quality.GOOD; case8_m.shutdownConfirmed := TRUE; case8_m.inRetracted := TRUE;
    CASE case8_phase OF
    0: case8_phase := 1;
    1: case8_m.command := E_ReferenceCommand.Home; case8_phase := 2;
    2: IF case8_m.sequence.State = TcForge.E_SM_State.READY THEN case8_phase := 3; END_IF;
    END_CASE;
ELSE
CASE case8_phase OF
3: case8_m.command := E_ReferenceCommand.Start; case8_phase := 4;
4:
    IF case8_m.outAdvance THEN case8_m.shutdownQuality := TcForge.E_IO_Quality.UNKNOWN; case8_m.command := E_ReferenceCommand.Abort; case8_phase := 5; END_IF;
5:
    AssertFalse(Condition := case8_m.outAdvance OR case8_m.outRetract, Message := 'Abort removes both coils');
    IF case8_age > 35 THEN
        AssertEquals_DINT(Expected := TcForge.E_SM_State.ABORTING, Actual := case8_m.sequence.State, Message := 'Untrusted feedback cannot confirm shutdown');
        case8_m.shutdownQuality := TcForge.E_IO_Quality.GOOD; case8_phase := 6;
    END_IF;
6:
    IF case8_m.sequence.State = TcForge.E_SM_State.STOPPED THEN case8_done := TRUE; END_IF;
END_CASE;
END_IF;
case8_m();
AssertFalse(Condition := case8_m.outAdvance AND case8_m.outRetract, Message := 'Coils must remain mutually exclusive');
case8_watchdog(IN := TRUE, PT := T#8S);
IF case8_watchdog.Q AND NOT case8_done THEN AssertTrue(Condition := FALSE, Message := 'Scenario did not reach its expected state'); case8_done := TRUE; END_IF;
IF case8_done THEN TEST_FINISHED(); END_IF;
END_METHOD

METHOD ResetRejectedDuringMotion
IF case9_done THEN RETURN; END_IF;
TEST('ResetRejectedDuringMotion');
case9_age := case9_age + 1;
case9_m.command := E_ReferenceCommand.None;
IF case9_phase < 3 THEN
    case9_m.inputQuality := TcForge.E_IO_Quality.GOOD; case9_m.outputQuality := TcForge.E_IO_Quality.GOOD;
    case9_m.shutdownQuality := TcForge.E_IO_Quality.GOOD; case9_m.shutdownConfirmed := TRUE; case9_m.inRetracted := TRUE;
    CASE case9_phase OF
    0: case9_phase := 1;
    1: case9_m.command := E_ReferenceCommand.Home; case9_phase := 2;
    2: IF case9_m.sequence.State = TcForge.E_SM_State.READY THEN case9_phase := 3; END_IF;
    END_CASE;
ELSE
CASE case9_phase OF
3: case9_m.command := E_ReferenceCommand.Start; case9_phase := 4;
4:
    IF case9_m.outAdvance THEN case9_m.command := E_ReferenceCommand.Reset; case9_phase := 5; END_IF;
5:
    AssertEquals_DINT(Expected := TcForge.E_RpcMethodResponse.REJECTED_WRONG_STATE, Actual := case9_m.lastResponse, Message := 'Reset during motion rejected');
    AssertTrue(Condition := case9_m.outAdvance AND NOT case9_m.faulted, Message := 'Rejected Reset must not alter the ongoing command');
    case9_m.command := E_ReferenceCommand.Abort;
    case9_done := TRUE;
END_CASE;
END_IF;
case9_m();
AssertFalse(Condition := case9_m.outAdvance AND case9_m.outRetract, Message := 'Coils must remain mutually exclusive');
case9_watchdog(IN := TRUE, PT := T#8S);
IF case9_watchdog.Q AND NOT case9_done THEN AssertTrue(Condition := FALSE, Message := 'Scenario did not reach its expected state'); case9_done := TRUE; END_IF;
IF case9_done THEN TEST_FINISHED(); END_IF;
END_METHOD

END_FUNCTION_BLOCK

// ---- Testing/Tests/FB_SequenceIntegrity_Test.TcPOU
FUNCTION_BLOCK FB_SequenceIntegrity_Test EXTENDS TcUnit.FB_TestSuite
VAR
    _done : BOOL;
    extraTimeout, extraZero, extraNegative, extraReset : TcForge.FB_Step;
    sm : FB_StateMachine_Probe;
    step_RejectNegativeDestination : TcForge.FB_Step;
    step_RejectOddDestination : TcForge.FB_Step;
    step_RejectCrossStateDestination : TcForge.FB_Step;
    step_RejectSelfDestination : TcForge.FB_Step;
    step_RejectNegativeTimeout : TcForge.FB_Step;
    step_TimeoutIncludesEntryAndSatisfiedConditions : TcForge.FB_Step;
    step_StopTimeoutEscalatesToAbort : TcForge.FB_Step;
    step_StopUserFaultEscalatesToAbort : TcForge.FB_Step;
    step_AbortTimeoutRequiresConfirmedShutdown : TcForge.FB_Step;
    step_CustomStepFaultCanRetry : TcForge.FB_Step;
    missing : TcForge.FB_StateMachine;
    duplicate : TcForge.FB_StateMachine;
    missingTarget : TcForge.FB_StateMachine;
    missingAbort : TcForge.FB_StateMachine;
    zero : TcForge.FB_StateMachine;
    duplicateA : TcForge.FB_Step;
    duplicateB : TcForge.FB_Step;
    targetStep : TcForge.FB_Step;
    zeroStep : TcForge.FB_Step;
END_VAR

IF _done THEN RETURN; END_IF;
RejectNegativeDestination();
RejectOddDestination();
RejectCrossStateDestination();
RejectSelfDestination();
RejectNegativeTimeout();
TimeoutIncludesEntryAndSatisfiedConditions();
StopTimeoutEscalatesToAbort();
StopUserFaultEscalatesToAbort();
AbortTimeoutRequiresConfirmedShutdown();
CustomStepFaultCanRetry();
MissingActiveStepFaults();
DuplicateActiveStepFaults();
MissingDestinationImplementationFaults();
MissingAbortImplementationFailsShutdown();
StepZeroNeverExecutes();
TimeoutAboveTimerRangeRejected();
ZeroFaultCodeStillInhibits();
NegativeFaultCodeStillInhibits();
InvalidResetPreservesShutdownLatch();
_done := TRUE;

METHOD RejectNegativeDestination
VAR

END_VAR
TEST('RejectNegativeDestination');
sm.ResetAll(); sm.ForceState(state := TcForge.E_SM_State.RUNNING); sm.SetCurrentStep(nStep := 3000);
step_RejectNegativeDestination(sm := sm, nStep := 3000, nNextStep := -2, nTimeout := 0);
AssertFalse(Condition := step_RejectNegativeDestination.Entry, Message := 'Invalid destination must inhibit Entry');
AssertEquals_DINT(Expected := TcForge.E_SM_Fault.InvalidStepConfiguration, Actual := sm.GetFaultCode(), Message := 'Configuration fault must be explicit');
TEST_FINISHED();
END_METHOD

METHOD RejectOddDestination
VAR

END_VAR
TEST('RejectOddDestination');
sm.ResetAll(); sm.ForceState(state := TcForge.E_SM_State.RUNNING); sm.SetCurrentStep(nStep := 3000);
step_RejectOddDestination(sm := sm, nStep := 3000, nNextStep := 3001, nTimeout := 0);
AssertFalse(Condition := step_RejectOddDestination.Entry, Message := 'Invalid destination must inhibit Entry');
AssertEquals_DINT(Expected := TcForge.E_SM_Fault.InvalidStepConfiguration, Actual := sm.GetFaultCode(), Message := 'Configuration fault must be explicit');
TEST_FINISHED();
END_METHOD

METHOD RejectCrossStateDestination
VAR

END_VAR
TEST('RejectCrossStateDestination');
sm.ResetAll(); sm.ForceState(state := TcForge.E_SM_State.RUNNING); sm.SetCurrentStep(nStep := 3000);
step_RejectCrossStateDestination(sm := sm, nStep := 3000, nNextStep := 5000, nTimeout := 0);
AssertFalse(Condition := step_RejectCrossStateDestination.Entry, Message := 'Invalid destination must inhibit Entry');
AssertEquals_DINT(Expected := TcForge.E_SM_Fault.InvalidStepConfiguration, Actual := sm.GetFaultCode(), Message := 'Configuration fault must be explicit');
TEST_FINISHED();
END_METHOD

METHOD RejectSelfDestination
VAR

END_VAR
TEST('RejectSelfDestination');
sm.ResetAll(); sm.ForceState(state := TcForge.E_SM_State.RUNNING); sm.SetCurrentStep(nStep := 3000);
step_RejectSelfDestination(sm := sm, nStep := 3000, nNextStep := 3000, nTimeout := 0);
AssertFalse(Condition := step_RejectSelfDestination.Entry, Message := 'Invalid destination must inhibit Entry');
AssertEquals_DINT(Expected := TcForge.E_SM_Fault.InvalidStepConfiguration, Actual := sm.GetFaultCode(), Message := 'Configuration fault must be explicit');
TEST_FINISHED();
END_METHOD

METHOD RejectNegativeTimeout
VAR

END_VAR
TEST('RejectNegativeTimeout');
sm.ResetAll(); sm.ForceState(state := TcForge.E_SM_State.RUNNING); sm.SetCurrentStep(nStep := 3000);
step_RejectNegativeTimeout(sm := sm, nStep := 3000, nNextStep := 3002, nTimeout := -1);
AssertFalse(Condition := step_RejectNegativeTimeout.Entry, Message := 'Negative timeout cannot silently disable protection');
AssertEquals_DINT(Expected := TcForge.E_SM_Fault.InvalidStepConfiguration, Actual := sm.GetFaultCode(), Message := 'Invalid timeout fault');
TEST_FINISHED();
END_METHOD

METHOD TimeoutIncludesEntryAndSatisfiedConditions
VAR

